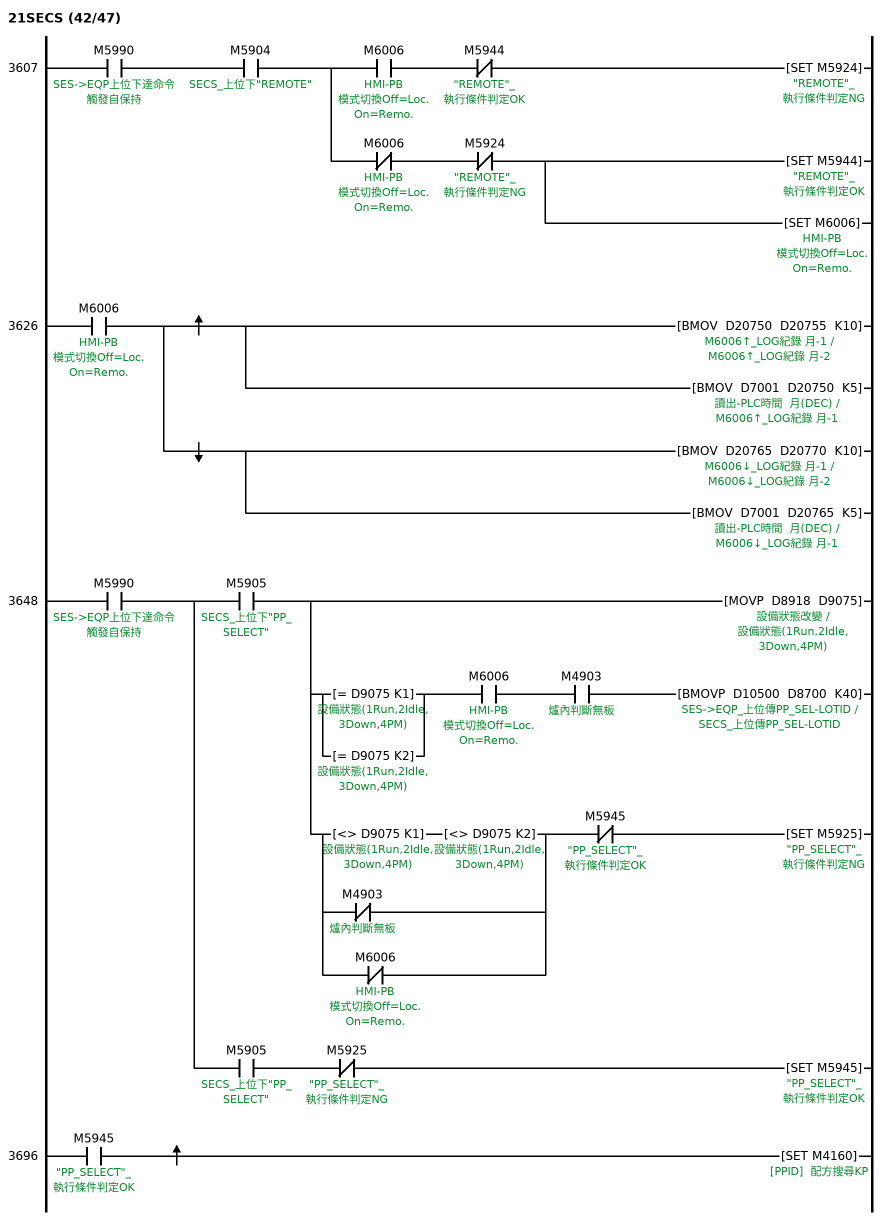
[picture p120: ladder of 21SECS, rungs at steps 3607 to 3696]
3607  LD      M5990  ; SES->EQP上位下達命令觸發自保持
      AND     M5904  ; SECS_上位下"REMOTE"
      MPS
      AND     M6006  ; HMI-PB  模式切換Off=Loc.On=Remo.
      ANI     M5944  ; "REMOTE"_執行條件判定OK
      SET     M5924  ; "REMOTE"_執行條件判定NG
        [note] "REMOTE CMD"
      MPP
      ANI     M6006  ; HMI-PB  模式切換Off=Loc.On=Remo.
      ANI     M5924  ; "REMOTE"_執行條件判定NG
      SET     M5944  ; "REMOTE"_執行條件判定OK
      SET     M6006  ; HMI-PB  模式切換Off=Loc.On=Remo.
3626  LD      M6006  ; HMI-PB  模式切換Off=Loc.On=Remo.
      MPS
      MEP
      BMOV    D20750 D20755 K10  ; M6006↑_LOG紀錄 月-1 / M6006↑_LOG紀錄 月-2
      BMOV    D7001 D20750 K5
      MPP
      MEF
      BMOV    D20765 D20770 K10  ; M6006↓_LOG紀錄 月-1 / M6006↓_LOG紀錄 月-2
      BMOV    D7001 D20765 K5
3648  LD      M5990  ; SES->EQP上位下達命令觸發自保持
      MPS
      AND     M5905  ; SECS_上位下"PP_SELECT"
      MOVP    D8918 D9075
        [note] "PP_SELECT CMD"
      MPS
      LD=     D9075 K1  ; 設備狀態(1Run,2Idle,3Down,4PM)
      OR=     D9075 K2  ; 設備狀態(1Run,2Idle,3Down,4PM)
      ANB
      AND     M6006  ; HMI-PB  模式切換Off=Loc.On=Remo.
      AND     M4903  ; 爐內判斷無板
      BMOVP   D10500 D8700 K40  ; SES->EQP_上位傳PP_SEL-LOTID / SECS_上位傳PP_SEL-LOTID
      MPP
      LD<>    D9075 K1  ; 設備狀態(1Run,2Idle,3Down,4PM)
      AND<>   D9075 K2  ; 設備狀態(1Run,2Idle,3Down,4PM)
      ORI     M4903  ; 爐內判斷無板
      ORI     M6006  ; HMI-PB  模式切換Off=Loc.On=Remo.
      ANB
      ANI     M5945  ; "PP_SELECT"_執行條件判定OK
      SET     M5925  ; "PP_SELECT"_執行條件判定NG
      MPP
      AND     M5905  ; SECS_上位下"PP_SELECT"
      ANI     M5925  ; "PP_SELECT"_執行條件判定NG
      SET     M5945  ; "PP_SELECT"_執行條件判定OK
3696  LD      M5945  ; "PP_SELECT"_執行條件判定OK
      MEP
      SET     M4160  ; [PPID]  配方搜尋KP
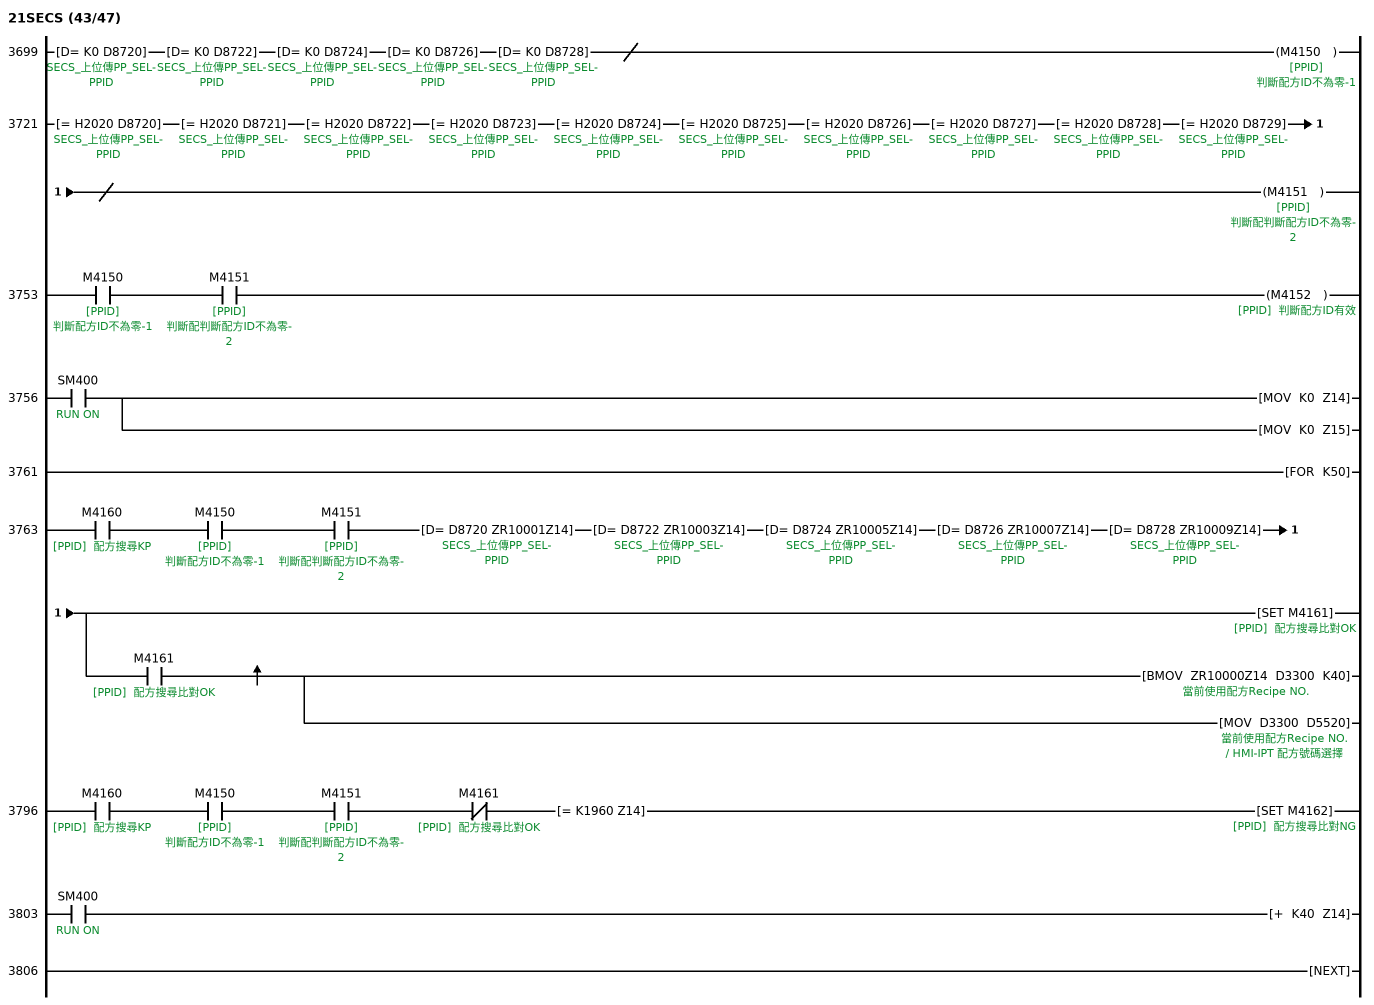
3699  LDD=    K0 D8720  ; SECS_上位傳PP_SEL-PPID
      ANDD=   K0 D8722  ; SECS_上位傳PP_SEL-PPID
      ANDD=   K0 D8724  ; SECS_上位傳PP_SEL-PPID
      ANDD=   K0 D8726  ; SECS_上位傳PP_SEL-PPID
      ANDD=   K0 D8728  ; SECS_上位傳PP_SEL-PPID
      INV
      OUT     M4150  ; [PPID]  判斷配方ID不為零-1
3721  LD=     H2020 D8720  ; SECS_上位傳PP_SEL-PPID
      AND=    H2020 D8721  ; SECS_上位傳PP_SEL-PPID
      AND=    H2020 D8722  ; SECS_上位傳PP_SEL-PPID
      AND=    H2020 D8723  ; SECS_上位傳PP_SEL-PPID
      AND=    H2020 D8724  ; SECS_上位傳PP_SEL-PPID
      AND=    H2020 D8725  ; SECS_上位傳PP_SEL-PPID
      AND=    H2020 D8726  ; SECS_上位傳PP_SEL-PPID
      AND=    H2020 D8727  ; SECS_上位傳PP_SEL-PPID
      AND=    H2020 D8728  ; SECS_上位傳PP_SEL-PPID
      AND=    H2020 D8729  ; SECS_上位傳PP_SEL-PPID
      INV
      OUT     M4151  ; [PPID]  判斷配判斷配方ID不為零-2
3753  LD      M4150  ; [PPID]  判斷配方ID不為零-1
      AND     M4151  ; [PPID]  判斷配判斷配方ID不為零-2
      OUT     M4152  ; [PPID]  判斷配方ID有效
3756  LD      SM400  ; RUN ON
      MOV     K0 Z14
      MOV     K0 Z15
3761  FOR     K50
3763  LD      M4160  ; [PPID]  配方搜尋KP
      AND     M4150  ; [PPID]  判斷配方ID不為零-1
      AND     M4151  ; [PPID]  判斷配判斷配方ID不為零-2
      ANDD=   D8720 ZR10001Z14  ; SECS_上位傳PP_SEL-PPID
      ANDD=   D8722 ZR10003Z14  ; SECS_上位傳PP_SEL-PPID
      ANDD=   D8724 ZR10005Z14  ; SECS_上位傳PP_SEL-PPID
      ANDD=   D8726 ZR10007Z14  ; SECS_上位傳PP_SEL-PPID
      ANDD=   D8728 ZR10009Z14  ; SECS_上位傳PP_SEL-PPID
      SET     M4161  ; [PPID]  配方搜尋比對OK
      AND     M4161  ; [PPID]  配方搜尋比對OK
      MEP
      BMOV    ZR10000Z14 D3300 K40
      MOV     D3300 D5520
3796  LD      M4160  ; [PPID]  配方搜尋KP
      AND     M4150  ; [PPID]  判斷配方ID不為零-1
      AND     M4151  ; [PPID]  判斷配判斷配方ID不為零-2
      ANI     M4161  ; [PPID]  配方搜尋比對OK
      AND=    K1960 Z14
      SET     M4162  ; [PPID]  配方搜尋比對NG
3803  LD      SM400  ; RUN ON
      +       K40 Z14
3806  NEXT
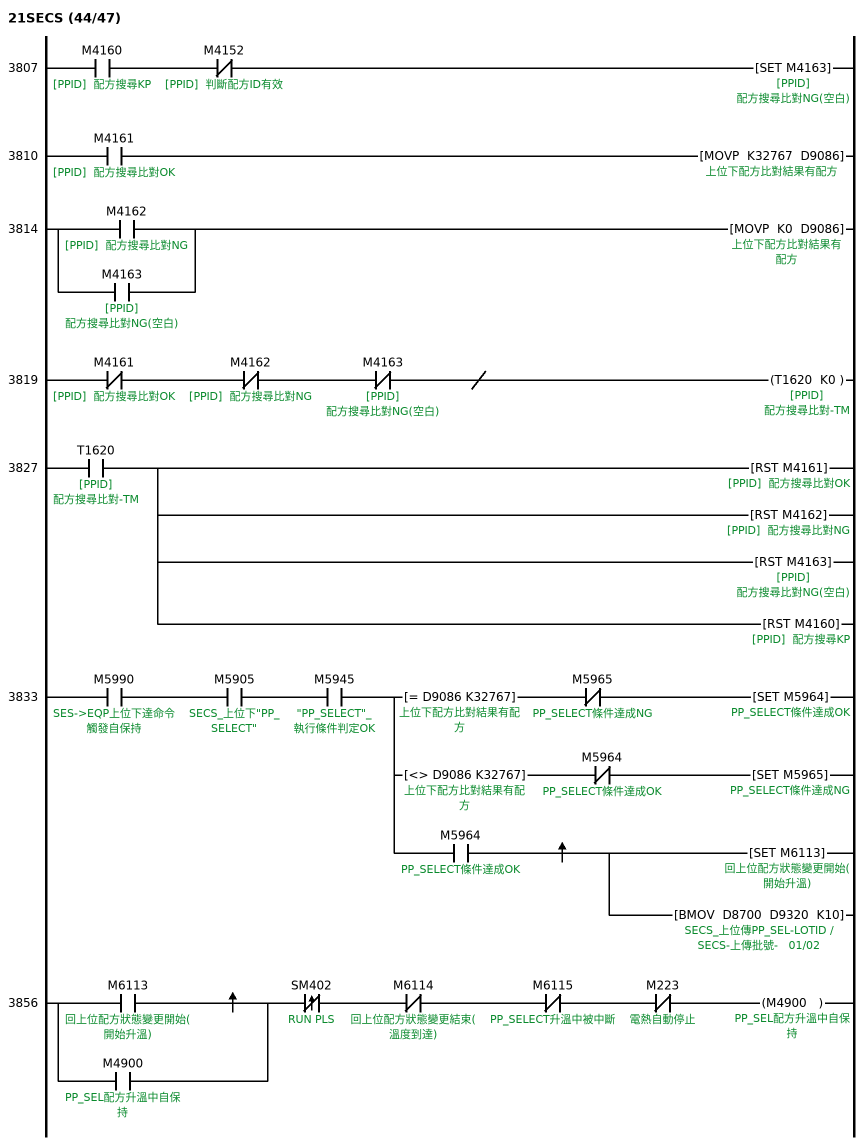
3807  LD      M4160  ; [PPID]  配方搜尋KP
      ANI     M4152  ; [PPID]  判斷配方ID有效
      SET     M4163  ; [PPID]  配方搜尋比對NG(空白)
3810  LD      M4161  ; [PPID]  配方搜尋比對OK
      MOVP    K32767 D9086
3814  LD      M4162  ; [PPID]  配方搜尋比對NG
      OR      M4163  ; [PPID]  配方搜尋比對NG(空白)
      MOVP    K0 D9086
3819  LDI     M4161  ; [PPID]  配方搜尋比對OK
      ANI     M4162  ; [PPID]  配方搜尋比對NG
      ANI     M4163  ; [PPID]  配方搜尋比對NG(空白)
      INV
      OUT     T1620 K0  ; [PPID]  配方搜尋比對-TM
3827  LD      T1620  ; [PPID]  配方搜尋比對-TM
      RST     M4161  ; [PPID]  配方搜尋比對OK
      RST     M4162  ; [PPID]  配方搜尋比對NG
      RST     M4163  ; [PPID]  配方搜尋比對NG(空白)
      RST     M4160  ; [PPID]  配方搜尋KP
3833  LD      M5990  ; SES->EQP上位下達命令觸發自保持
      AND     M5905  ; SECS_上位下"PP_SELECT"
      AND     M5945  ; "PP_SELECT"_執行條件判定OK
      MPS
      AND=    D9086 K32767  ; 上位下配方比對結果有配方
      ANI     M5965  ; PP_SELECT條件達成NG
      SET     M5964  ; PP_SELECT條件達成OK
      MRD
      AND<>   D9086 K32767  ; 上位下配方比對結果有配方
      ANI     M5964  ; PP_SELECT條件達成OK
      SET     M5965  ; PP_SELECT條件達成NG
      MPP
      AND     M5964  ; PP_SELECT條件達成OK
      MEP
      SET     M6113  ; 回上位配方狀態變更開始(開始升溫)
      BMOV    D8700 D9320 K10  ; SECS-上傳批號-   01/02
3856  LD      M6113  ; 回上位配方狀態變更開始(開始升溫)
      MEP
      OR      M4900  ; PP_SEL配方升溫中自保持
      ANDPI   SM402  ; RUN PLS
      ANI     M6114  ; 回上位配方狀態變更結束(溫度到達)
      ANI     M6115  ; PP_SELECT升溫中被中斷
      ANI     M223  ; 電熱自動停止
      OUT     M4900  ; PP_SEL配方升溫中自保持
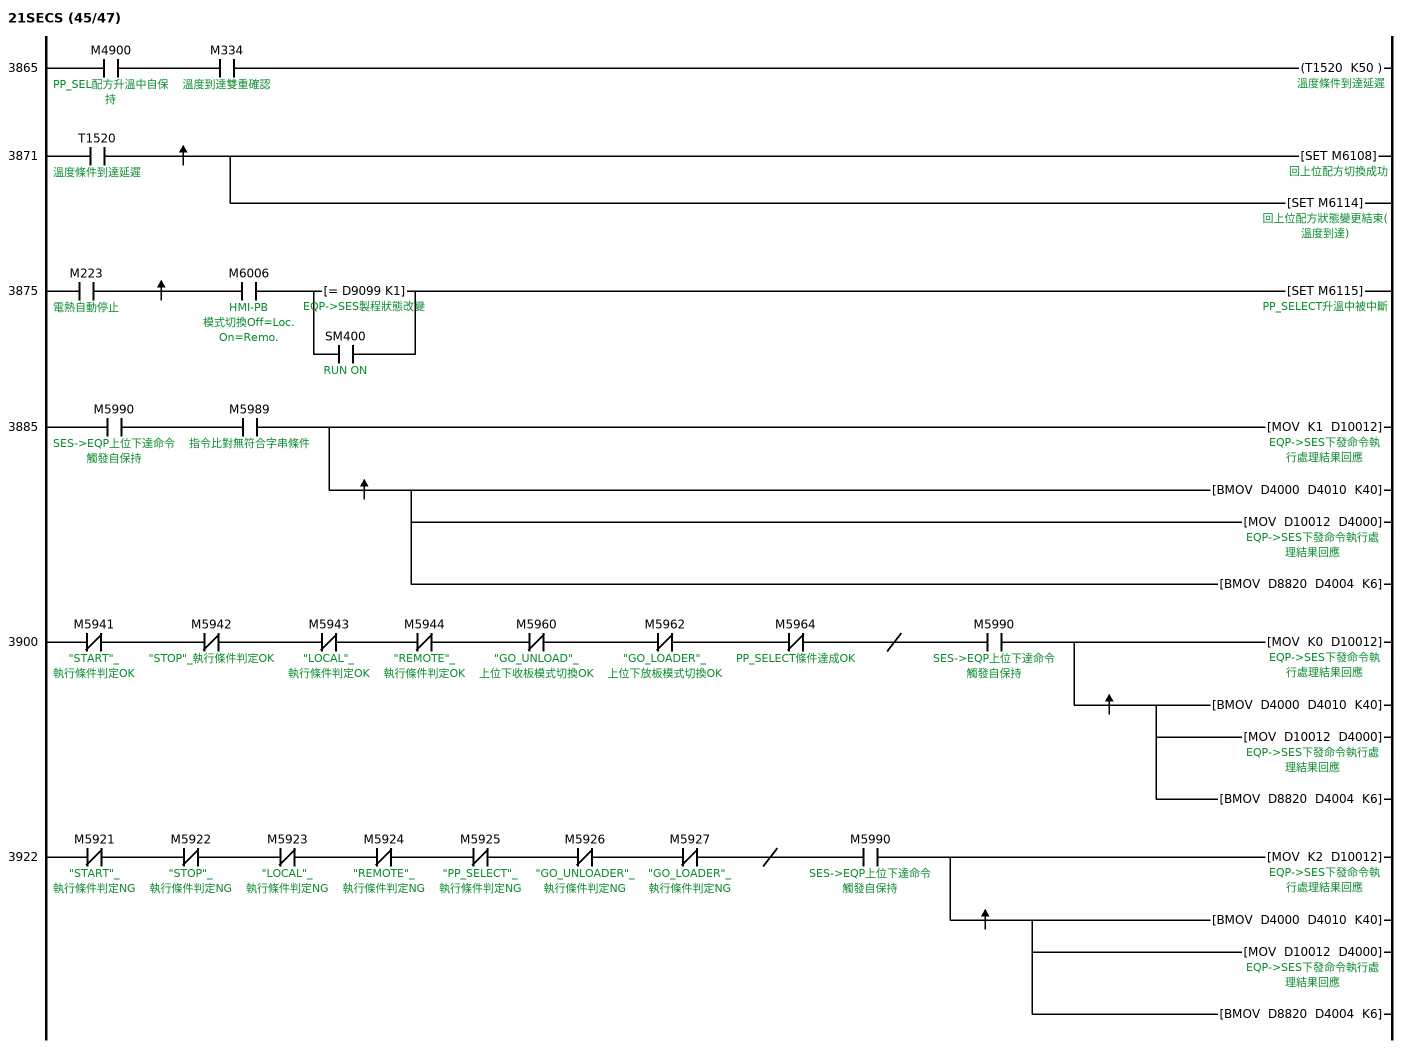
3865  LD      M4900  ; PP_SEL配方升溫中自保持
      AND     M334  ; 溫度到達雙重確認
      OUT     T1520 K50  ; 溫度條件到達延遲
3871  LD      T1520  ; 溫度條件到達延遲
      MEP
      SET     M6108  ; 回上位配方切換成功
      SET     M6114  ; 回上位配方狀態變更結束(溫度到達)
3875  LD      M223  ; 電熱自動停止
      MEP
      AND     M6006  ; HMI-PB  模式切換Off=Loc.On=Remo.
      LD=     D9099 K1  ; EQP->SES製程狀態改變
      OR      SM400  ; RUN ON
      ANB
      SET     M6115  ; PP_SELECT升溫中被中斷
3885  LD      M5990  ; SES->EQP上位下達命令觸發自保持
      AND     M5989  ; 指令比對無符合字串條件
      MOV     K1 D10012
      MEP
      BMOV    D4000 D4010 K40
      MOV     D10012 D4000
      BMOV    D8820 D4004 K6
3900  LDI     M5941  ; "START"_執行條件判定OK
      ANI     M5942  ; "STOP"_執行條件判定OK
      ANI     M5943  ; "LOCAL"_執行條件判定OK
      ANI     M5944  ; "REMOTE"_執行條件判定OK
      ANI     M5960  ; "GO_UNLOAD"_上位下收板模式切換OK
      ANI     M5962  ; "GO_LOADER"_上位下放板模式切換OK
      ANI     M5964  ; PP_SELECT條件達成OK
      INV
      AND     M5990  ; SES->EQP上位下達命令觸發自保持
      MOV     K0 D10012
      MEP
      BMOV    D4000 D4010 K40
      MOV     D10012 D4000
      BMOV    D8820 D4004 K6
3922  LDI     M5921  ; "START"_執行條件判定NG
      ANI     M5922  ; "STOP"_執行條件判定NG
      ANI     M5923  ; "LOCAL"_執行條件判定NG
      ANI     M5924  ; "REMOTE"_執行條件判定NG
      ANI     M5925  ; "PP_SELECT"_執行條件判定NG
      ANI     M5926  ; "GO_UNLOADER"_執行條件判定NG
      ANI     M5927  ; "GO_LOADER"_執行條件判定NG
      INV
      AND     M5990  ; SES->EQP上位下達命令觸發自保持
      MOV     K2 D10012
      MEP
      BMOV    D4000 D4010 K40
      MOV     D10012 D4000
      BMOV    D8820 D4004 K6
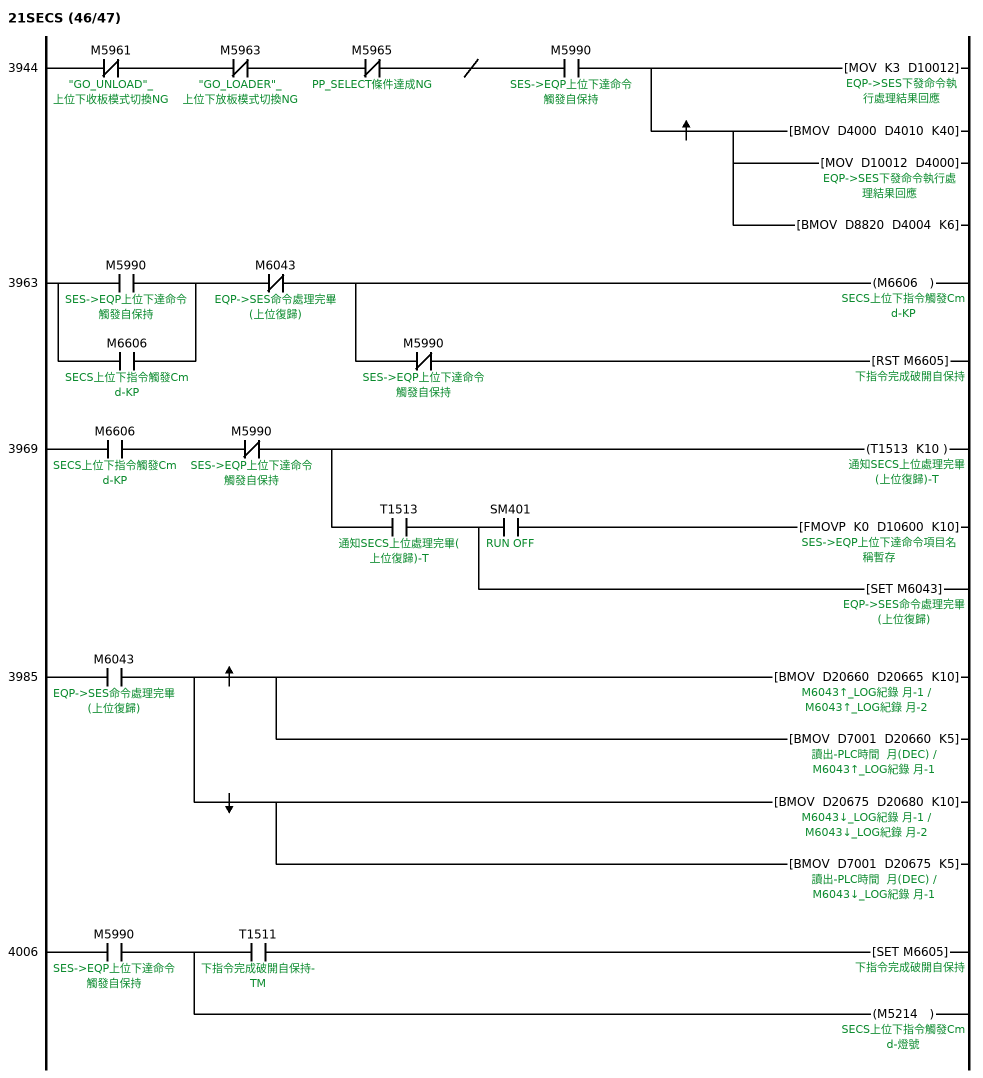
3944  LDI     M5961  ; "GO_UNLOAD"_上位下收板模式切換NG
      ANI     M5963  ; "GO_LOADER"_上位下放板模式切換NG
      ANI     M5965  ; PP_SELECT條件達成NG
      INV
      AND     M5990  ; SES->EQP上位下達命令觸發自保持
      MOV     K3 D10012
      MEP
      BMOV    D4000 D4010 K40
      MOV     D10012 D4000
      BMOV    D8820 D4004 K6
3963  LD      M5990  ; SES->EQP上位下達命令觸發自保持
      OR      M6606  ; SECS上位下指令觸發Cmd-KP
      ANI     M6043  ; EQP->SES命令處理完畢(上位復歸)
      OUT     M6606  ; SECS上位下指令觸發Cmd-KP
      ANI     M5990  ; SES->EQP上位下達命令觸發自保持
      RST     M6605  ; 下指令完成破開自保持
3969  LD      M6606  ; SECS上位下指令觸發Cmd-KP
      ANI     M5990  ; SES->EQP上位下達命令觸發自保持
      OUT     T1513 K10  ; 通知SECS上位處理完畢(上位復歸)-T
      AND     T1513  ; 通知SECS上位處理完畢(上位復歸)-T
      MPS
      AND     SM401  ; RUN OFF
      FMOVP   K0 D10600 K10
      MPP
      SET     M6043  ; EQP->SES命令處理完畢(上位復歸)
3985  LD      M6043  ; EQP->SES命令處理完畢(上位復歸)
      MPS
      MEP
      BMOV    D20660 D20665 K10  ; M6043↑_LOG紀錄 月-1 / M6043↑_LOG紀錄 月-2
      BMOV    D7001 D20660 K5
      MPP
      MEF
      BMOV    D20675 D20680 K10  ; M6043↓_LOG紀錄 月-1 / M6043↓_LOG紀錄 月-2
      BMOV    D7001 D20675 K5
4006  LD      M5990  ; SES->EQP上位下達命令觸發自保持
      MPS
      AND     T1511  ; 下指令完成破開自保持-TM
      SET     M6605  ; 下指令完成破開自保持
      MPP
      OUT     M5214  ; SECS上位下指令觸發Cmd-燈號
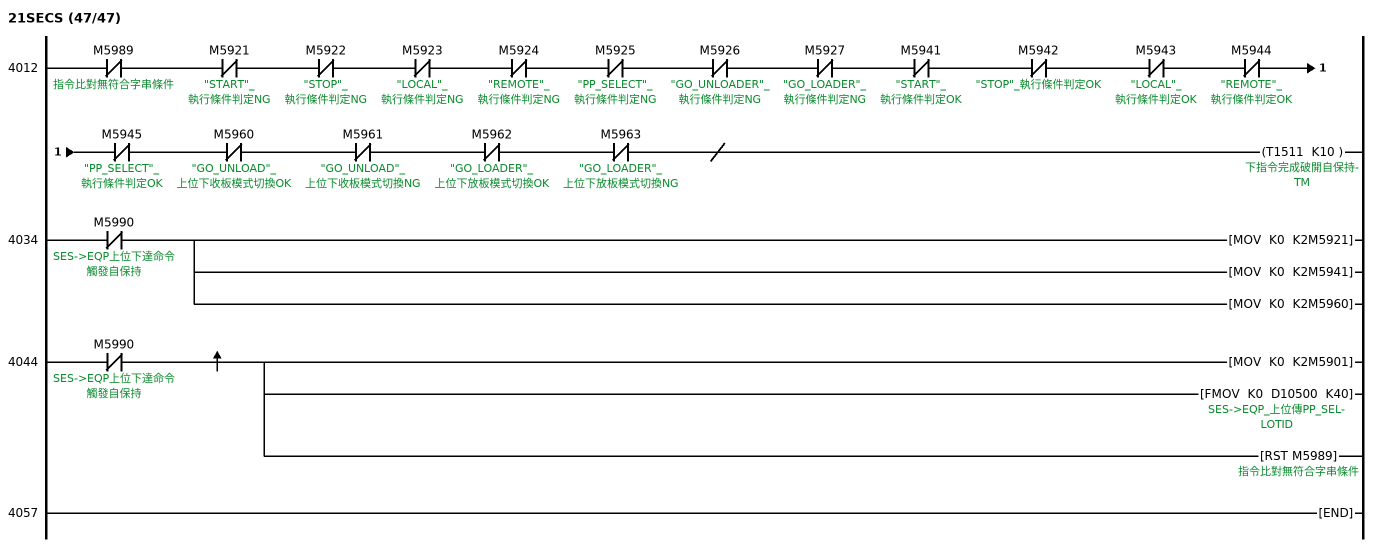
4012  LDI     M5989  ; 指令比對無符合字串條件
      ANI     M5921  ; "START"_執行條件判定NG
      ANI     M5922  ; "STOP"_執行條件判定NG
      ANI     M5923  ; "LOCAL"_執行條件判定NG
      ANI     M5924  ; "REMOTE"_執行條件判定NG
      ANI     M5925  ; "PP_SELECT"_執行條件判定NG
      ANI     M5926  ; "GO_UNLOADER"_執行條件判定NG
      ANI     M5927  ; "GO_LOADER"_執行條件判定NG
      ANI     M5941  ; "START"_執行條件判定OK
      ANI     M5942  ; "STOP"_執行條件判定OK
      ANI     M5943  ; "LOCAL"_執行條件判定OK
      ANI     M5944  ; "REMOTE"_執行條件判定OK
      ANI     M5945  ; "PP_SELECT"_執行條件判定OK
      ANI     M5960  ; "GO_UNLOAD"_上位下收板模式切換OK
      ANI     M5961  ; "GO_UNLOAD"_上位下收板模式切換NG
      ANI     M5962  ; "GO_LOADER"_上位下放板模式切換OK
      ANI     M5963  ; "GO_LOADER"_上位下放板模式切換NG
      INV
      OUT     T1511 K10  ; 下指令完成破開自保持-TM
4034  LDI     M5990  ; SES->EQP上位下達命令觸發自保持
      MOV     K0 K2M5921
      MOV     K0 K2M5941
      MOV     K0 K2M5960
4044  LDI     M5990  ; SES->EQP上位下達命令觸發自保持
      MEP
      MOV     K0 K2M5901
      FMOV    K0 D10500 K40
      RST     M5989  ; 指令比對無符合字串條件
4057  END
END_PROGRAM

// device comments not shown above
X4  ; 手動放板夾爪--放定點
X5  ; 手動放板夾爪--夾定點
X11  ; 取板完成位(連線)
X14  ; 下料旋臂長程中定點
X3C  ; 進料ROBOT左真空檢知
X7E  ; 印刷機出板要求
X332  ; FR1-DO(31)
X333  ; FR1-DO(32)
X334  ; FR1-DO(33)
X335  ; FR1-DO(34)
X336  ; FR1-DO(35)
X337  ; FR1-DO(36)
X338  ; FR1-DO(37)
X339  ; FR1-DO(38)
X33A  ; FR1-DO(39)
X33B  ; FR1-DO(40)
X33C  ; FR1-DO(41)
X33D  ; FR1-DO(42)
X33E  ; FR1-DO(43)
X33F  ; FR1-DO(44)
X340  ; FR1-DO(45)
X341  ; FR1-DO(46)
X342  ; FR1-DO(47)
X343  ; FR1-DO(48)
X344  ; FR1-DO(49)
X345  ; FR1-DO(50)
X346  ; FR1-DO(51)
X347  ; FR1-DO(52)
X348  ; FR1-DO(53)
X349  ; FR1-DO(54)
X34A  ; FR1-DO(55)
X34B  ; FR1-DO(56)
X34C  ; FR1-DO(57)
X34D  ; FR1-DO(58)
X34E  ; FR1-DO(59)
X34F  ; FR1-DO(60)
X350  ; FR1-DO(61)
X351  ; FR1-DO(62)
X352  ; FR1-DO(63)
X353  ; FR1-DO(64)
X354  ; FR1-DO(65)
X355  ; FR1-DO(66)
X356  ; FR1-DO(67)
X357  ; FR1-DO(68)
X358  ; FR1-DO(69)
X359  ; FR1-DO(70)
X35A  ; FR1-DO(71)
X35B  ; FR1-DO(72)
X35C  ; FR1-DO(73)
X35D  ; FR1-DO(74)
X35E  ; FR1-DO(75)
X35F  ; FR1-DO(76)
X360  ; FR1-DO(77)
X361  ; FR1-DO(78)
X362  ; FR1-DO(79)
X363  ; FR1-DO(80)
X364  ; FR1-DO(81)
X365  ; FR1-DO(82)
X366  ; FR1-DO(83)
X367  ; FR1-DO(84)
X368  ; FR1-DO(85)
X369  ; FR1-DO(86)
X36A  ; FR1-DO(87)
X36B  ; FR1-DO(88)
X36C  ; FR1-DO(89)
X36D  ; FR1-DO(90)
X36E  ; FR1-DO(91)
X36F  ; FR1-DO(92)
X370  ; FR1-DO(93)
X371  ; FR1-DO(94)
X372  ; FR1-DO(95)
X373  ; FR1-DO(96)
X374  ; FR1-DO(97)
X375  ; FR1-DO(98)
X376  ; FR1-DO(99)
X377  ; FR1-DO(100)
X378  ; FR1-DO(101)
X379  ; FR1-DO(102)
X37A  ; FR1-DO(103)
X37B  ; FR1-DO(104)
X37C  ; FR1-DO(105)
X37D  ; FR1-DO(106)
X37E  ; FR1-DO(107)
X37F  ; FR1-DO(108)
X0A03  ; Other station   DataLinkStatus
X1302  ; <印刷機>異常
Y10C  ; 進料連線--取板完
Y122  ; 進料ROBOT左真空SV
Y123  ; 進料ROBOT右真空SV
Y320  ; ROBOT GO HOME
Y330  ; TR1-DI(31)
Y331  ; TR1-DI(32)
Y332  ; TR1-DI(33)
Y333  ; TR1-DI(34)
Y334  ; TR1-DI(35)
Y335  ; TR1-DI(36)
Y336  ; TR1-DI(37)
Y337  ; TR1-DI(38)
Y338  ; TR1-DI(39)
Y339  ; TR1-DI(40)
Y33A  ; TR1-DI(41)
Y33B  ; TR1-DI(42)
Y33C  ; TR1-DI(43)
Y33D  ; TR1-DI(44)
Y33E  ; TR1-DI(45)
Y33F  ; TR1-DI(46)
Y340  ; TR1-DI(47)
Y341  ; TR1-DI(48)
Y342  ; TR1-DI(49)
Y343  ; TR1-DI(50)
Y344  ; TR1-DI(51)
Y345  ; TR1-DI(52)
Y346  ; TR1-DI(53)
Y347  ; TR1-DI(54)
Y348  ; TR1-DI(55)
Y349  ; TR1-DI(56)
Y34A  ; TR1-DI(57)
Y34B  ; TR1-DI(58)
Y34C  ; TR1-DI(59)
Y34D  ; TR1-DI(60)
Y34E  ; TR1-DI(61)
Y34F  ; TR1-DI(62)
Y350  ; TR1-DI(63)
Y351  ; TR1-DI(64)
Y352  ; TR1-DI(65)
Y353  ; TR1-DI(66)
Y354  ; TR1-DI(67)
Y355  ; TR1-DI(68)
Y356  ; TR1-DI(69)
Y357  ; TR1-DI(70)
Y358  ; TR1-DI(71)
Y359  ; TR1-DI(72)
Y35A  ; TR1-DI(73)
Y35B  ; TR1-DI(74)
Y35C  ; TR1-DI(75)
Y35D  ; TR1-DI(76)
Y35E  ; TR1-DI(77)
Y35F  ; TR1-DI(78)
Y360  ; TR1-DI(79)
Y361  ; TR1-DI(80)
Y362  ; TR1-DI(81)
Y363  ; TR1-DI(82)
Y364  ; TR1-DI(83)
Y365  ; TR1-DI(84)
Y366  ; TR1-DI(85)
Y367  ; TR1-DI(86)
Y368  ; TR1-DI(87)
Y369  ; TR1-DI(88)
Y36A  ; TR1-DI(89)
Y36B  ; TR1-DI(90)
Y36C  ; TR1-DI(91)
Y36D  ; TR1-DI(92)
Y36E  ; TR1-DI(93)
Y36F  ; TR1-DI(94)
Y370  ; TR1-DI(95)
Y371  ; TR1-DI(96)
Y372  ; TR1-DI(97)
Y373  ; TR1-DI(98)
Y374  ; TR1-DI(99)
Y375  ; TR1-DI(100)
Y376  ; TR1-DI(101)
Y377  ; TR1-DI(102)
Y378  ; TR1-DI(103)
Y379  ; TR1-DI(104)
Y37A  ; TR1-DI(105)
Y37B  ; TR1-DI(106)
Y37C  ; TR1-DI(107)
Y37D  ; TR1-DI(108)
Y37E  ; TR1-DI(109)
Y37F  ; TR1-DI(110)
M40  ; 手動放板側邊上料_放板PB
M42  ; 夾爪開爪腳踏開關_側邊上料使用PB
M55  ; 板材尺寸連線/本機模式PB
M70  ; 昇降上昇位置教導設定PB
M71  ; 昇降上等待位置教導設定PB
M73  ; 昇降下降位置教導設定PB
M76  ; 下料鼓風機自動
M79  ; 下料鼓風機手動
M140  ; 手動放板側邊上料_放板燈
M141  ; 手動放板側邊上料_夾板燈
M182  ; 進料照明開
M185  ; 出料照明開
M190  ; 上料掉板後原點復歸
M191  ; 上料掉板後原點復歸STOP
M221  ; 搬移停止
M234  ; 自動模式鏈條拉緊PLS
M237  ; 上料夾爪可伸出KP
M316  ; 開機鏈條張力自動拉緊
M317  ; 鏈條張力拉緊KP
M318  ; 主傳動步進拉緊
M324  ; 電熱溫度到達KP
M325  ; 電熱溫度到達計時
M326  ; 開機計時24小時到
M327  ; 油壓張力檢知
M332  ; 進料輸送停止
M333  ; 進料輸送減速KP
M335  ; 升溫中狀態
M375  ; 手動放板側邊上料_放板
M376  ; 手動放板側邊上料_夾板
M377  ; 手動上板PB4指示燈
M439  ; 進料ROBOT禁止回原點
M514  ; 下料旋臂長程中定點
M552  ; 進料集塵鼓風機手動運轉
M553  ; 出料集塵鼓風機手動運轉
M554  ; 進出料集塵鼓風機自動運轉
M595  ; #06 風車PB
M596  ; #07 風車PB
M597  ; #08 風車PB
M598  ; #09 風車PB
M599  ; #10 風車PB
M600  ; #11 風車PB
M601  ; #12 風車PB
M602  ; #13 風車PB
M603  ; #14 風車PB
M604  ; #15 風車PB
M605  ; #16 風車PB
M606  ; #17 風車PB
M615  ; #06 電熱PB
M616  ; #07 電熱PB
M617  ; #08 電熱PB
M618  ; #09 電熱PB
M619  ; #10 電熱PB
M620  ; #11 電熱PB
M621  ; #12 電熱PB
M622  ; #13 電熱PB
M623  ; #14 電熱PB
M624  ; #15 電熱PB
M625  ; #16 電熱PB
M626  ; #17 電熱PB
M700  ; SECS_USE清除進板訊號
M701  ; SECS_USE進板訊號ON
M725  ; #06 風車訊號
M726  ; #07 風車訊號
M727  ; #08 風車訊號
M728  ; #09 風車訊號
M729  ; #10 風車訊號
M730  ; #11 風車訊號
M731  ; #12 風車訊號
M732  ; #13 風車訊號
M733  ; #14 風車訊號
M734  ; #15 風車訊號
M735  ; #16 風車訊號
M736  ; #17 風車訊號
M785  ; #06 電熱訊號
M786  ; #07 電熱訊號
M787  ; #08 電熱訊號
M788  ; #09 電熱訊號
M789  ; #10 電熱訊號
M790  ; #11 電熱訊號
M791  ; #12 電熱訊號
M792  ; #13 電熱訊號
M793  ; #14 電熱訊號
M794  ; #15 電熱訊號
M795  ; #16 電熱訊號
M796  ; #17 電熱訊號
M805  ; 上料夾爪短程縮回KP
M825  ; #06 溫度到達KP
M826  ; #07 溫度到達KP
M827  ; #08 溫度到達KP
M828  ; #09 溫度到達KP
M829  ; #10 溫度到達KP
M830  ; #11 溫度到達KP
M831  ; #12 溫度到達KP
M832  ; #13 溫度到達KP
M833  ; #14 溫度到達KP
M834  ; #15 溫度到達KP
M835  ; #16 溫度到達KP
M836  ; #17 溫度到達KP
M1010  ; SECS_USE指令比對正確
M1011  ; PP_SELECT條件達成
M1304  ; 進料段無板
M1305  ; 進料定位有板
M1518  ; 風車停止備用1PLS
M1519  ; 風車停止備用2PLS
M1605  ; #06 電熱AL2 超溫
M1606  ; #07 電熱AL2 超溫
M1607  ; #08 電熱AL2 超溫
M1615  ; 冷卻段電熱AL2 超溫
M1621  ; #06 電熱OTP 超溫
M1622  ; #07 電熱OTP 超溫
M1623  ; #08 電熱OTP 超溫
M1637  ; #06 風車過載
M1638  ; #07 風車過載
M1639  ; #08 風車過載
M1653  ; #06 低溫警報
M1654  ; #07 低溫警報
M1655  ; #08 低溫警報
M4704  ; 生產片數到達
M4713  ; 拍板馬達伺服運轉逾時異常
M4716  ; 拍板馬達伺服內極限
M4717  ; 拍板馬達伺服外極限
M4917  ; 刪除配方名稱
M4920  ; 入口計數
M4921  ; 出口計數
M4922  ; 爐內限制異常
M4923  ; 出口計數
M4925  ; 卡板不警報
M4930  ; 點燈運轉KP
M4931  ; 點燈停止
M4932  ; 上位下啟動訊號
M4933  ; PP_SELECT點燈用保持
M4934  ; 上位允許放板START
M4935  ; 上位下暫停進板
M4936  ; HMI-Show_SEC模式未START
M4937  ; 上位要儲存配方
M4943  ; 上位下GO_REMOTE
M4944  ; 上位下GO-LOCAL
M4945  ; 上位允許放板START保持
M4950  ; 點燈中請稍待指示
M4951  ; 熄點燈冷卻中請稍待指示
M4953  ; 熄燈OK狀態
M4956  ; 輸送機停止熄燈
M4990  ; 密碼ENT
M4992  ; 密碼ENT Keep
M4993  ; 參數設定取消PB
M4994  ; 參數設定取消PLS
M4996  ; 離線測試用
M4999  ; 回上位生產停止
M5004  ; ##未完成生產片數到達
M5034  ; 輸送運轉未加熱完成
M5075  ; 回上位生產完成保持
M5076  ; IDLE-   FLAG
M5101  ; 三色紅燈
M5102  ; 三色綠燈
M5106  ; 未知?測試用
M5203  ; 未知?測試用
M5204  ; 上位允許放板START
M5205  ; 上位停止放板並清出料號
M5206  ; 上位下配方和啟動輸送和點燈
M5207  ; 上位切換成GO-REMOTE
M5208  ; 上位切換成GO-LOCAL
M5209  ; 上位下暫停進板
M5210  ; 上位下恢復進板
M5213  ; 上位下指令觸發bit
M5215  ; Barcod啟動固定式完成
M5216  ; 上位字串比對不對(開始,停止,配方)
M5217  ; 門,(1)(2),PPID,配方名稱比對不對
M5314  ; 配方刪除
M5315  ; 配方儲存
M5316  ; 呼叫Q的配方
M5317  ; 比對配方用
M5318  ; 自動
M5319  ; 手動
M5320  ; FX機台狀態改變
M5321  ; 自動啟動
M5322  ; 程式結束
M5323  ; 緊急停止開關
M5325  ; 對話視窗關閉
M5326  ; 配方新增
M5327  ; 配方修改
M5328  ; 配方刪除
M5329  ; 機構異常警報
M5347  ; 配方Barcode掃描
M5348  ; 工單輸入
M5349  ; Barcod啟動固定式
M5350  ; Bey Pass PB
M5351  ; 自動PB
M5352  ; 連線開放OP控制
M5353  ; 確認(101頁)人機SET
M5354  ; 確認(102頁)人機SET
M5410  ; [ES-01] GREEN_  LiGHT   OFF
M5411  ; [ES-01] GREEN_  LiGHT   ON
M5412  ; [ES-01] GREEN_  LiGHT   FLASH
M5413  ; [ES-01] RED_    LiGHT   OFF
M5414  ; [ES-01] RED_    LiGHT   ON
M5415  ; [ES-01] RED_    LiGHT   FLASH
M5416  ; [ES-01] YELLOW_ LiGHT   OFF
M5417  ; [ES-01] YELLOW_ LiGHT   ON
M5418  ; [ES-01] YELLOW_ LiGHT   FLASH
M5928  ; "STC"_執行條件判定NG
M5929  ; "BUZZER"_執行條件判定NG
M5946  ; "GO_UNLOADER"_執行條件判定OK
M5947  ; "GO_LOADER"_執行條件判定OK
M5948  ; "STC"_執行條件判定OK
M5949  ; "BUZZER"_執行條件判定OK
M5970  ; MES收板模式初始化動作中
M5972  ; MES放板模式初始化動作中
M6140  ; 要求上位回讀工單板號右爐
M6141  ; 要求上位回讀工單右爐
M6231  ; 上位要儲存配方
M6600  ; SECS上位下指令觸發Cmd-KP
M6607  ; Host刪除配方自保持
M6608  ; Host刪除配方自清除保持
M6610  ; 比對M700~M715都等於零
M6611  ; 比對M716~M731都等於零
M6820  ; 比對GO-REMOTE字串不對
M6821  ; 名稱GO-LOCAL比對不對
M6822  ; 比對RESUME字串不對
M6823  ; 比對PPID字串不對
M6824  ; 比對PAUSE字串不對
M6825  ; 比對START字串不對
M6826  ; 比對STOP字串不對
M6827  ; 比對PP_SELECT字串不對
M6854  ; 機台再IDEL
M6860  ; 機台不在可生產狀態
M6861  ; 下STOP 機台不再READY/EXECUTING
M6862  ; 下PP_SELECT 機台不在待機中(IDLE)
M6863  ; 設備沒再暫停狀態
M6864  ; 機台不再START 狀態
M6865  ; 機台狀態不對
M6866  ; 設備沒再LOCAL狀態
M6867  ; 設備沒再REMOTE狀態
M6999  ; 三色綠燈
M7001  ; 三色紅燈
M7012  ; 回應HOST要儲存配方同步
M7014  ; 回應HOST刪除配方同步
M7600  ; RUN ON
L3804  ; 第05站  CC-LINK 異常
L3805  ; 第06站  CC-LINK 異常
L3806  ; 第07站  CC-LINK 異常
L3807  ; 第08站  CC-LINK 異常
L3808  ; 第09站  CC-LINK 異常
L3809  ; 第10站  CC-LINK 異常
L3810  ; 第11站  CC-LINK 異常
L3811  ; 第12站  CC-LINK 異常
L3812  ; 第13站  CC-LINK 異常
L3813  ; 第14站  CC-LINK 異常
L3814  ; 第15站  CC-LINK 異常
L3815  ; 第16站  CC-LINK 異常
T8  ; 上料伺服自動復歸次數未到計時
T11  ; 上料伺服自動復歸計時
T12  ; 上料手臂夾爪夾自動延遲
T13  ; 上料昇降伺服運轉延遲
T16  ; 昇降上昇位置教導延遲
T17  ; 昇降上等待位置教導延遲
T19  ; 昇降下降位置教導延遲
T39  ; 下料鼓風機自動停止
T47  ; 進料集塵鼓風機PB延遲
T48  ; 出料集塵鼓風機PB延遲
T49  ; 集塵鼓風機運轉停止延遲
T54  ; 進料段無板延遲
T56  ; ROBOT外部循環啟動計時
T68  ; 進料輸送減速光電延遲
T75  ; 油壓馬達送電前進10秒
T105  ; #06 風車PB延遲
T106  ; #07 風車PB延遲
T107  ; #08 風車PB延遲
T108  ; #09 風車PB延遲
T109  ; #10 風車PB延遲
T110  ; #11 風車PB延遲
T111  ; #12 風車PB延遲
T112  ; #13 風車PB延遲
T113  ; #14 風車PB延遲
T114  ; #15 風車PB延遲
T115  ; #16 風車PB延遲
T116  ; #17 風車PB延遲
T125  ; #06 電熱PB延遲
T126  ; #07 電熱PB延遲
T127  ; #08 電熱PB延遲
T128  ; #09 電熱PB延遲
T129  ; #10 電熱PB延遲
T130  ; #11 電熱PB延遲
T131  ; #12 電熱PB延遲
T132  ; #13 電熱PB延遲
T133  ; #14 電熱PB延遲
T134  ; #15 電熱PB延遲
T135  ; #16 電熱PB延遲
T136  ; #17 電熱PB延遲
T139  ; #17 低溫警報
T145  ; #06 低溫警報
T146  ; #07 低溫警報
T147  ; #08 低溫警報
T148  ; #09 低溫警報
T149  ; #10 低溫警報
T150  ; #11 低溫警報
T151  ; #12 低溫警報
T152  ; #13 低溫警報
T159  ; 進料輸送夾爪夾板異常延遲
T163  ; 進料輸送垂直異常延遲
T164  ; 進料輸送水平異常延遲
T165  ; 上料夾爪長程伸異常延遲
T166  ; 上料夾爪長程縮異常延遲
T186  ; 油壓馬達運轉計時
T188  ; 進料輸送運轉逾時
T190  ; 進料輸送掉板異常延遲
T191  ; 上料夾爪掉板異常延遲
T196  ; 進料空氣壓力異常延時
T200  ; 進料輸送停止時間延遲
T204  ; 進料ROBOT左真空檢知異常TM
T205  ; 進料ROBOT右真空檢知異常TM
T208  ; 手動上板檢知光電異常TM
T400  ; #01 風車INV運轉計時
T401  ; #02 風車INV運轉計時
T402  ; #03 風車INV運轉計時
T403  ; #04 風車INV運轉計時
T404  ; #05 風車INV運轉計時
T405  ; #06 風車INV運轉計時
T406  ; #07 風車INV運轉計時
T407  ; #08 風車INV運轉計時
T408  ; #09 風車INV運轉計時
T409  ; #10 風車INV運轉計時
T410  ; #11 風車INV運轉計時
T411  ; #12 風車INV運轉計時
T412  ; #13 風車INV運轉計時
T413  ; #14 風車INV運轉計時
T414  ; #15 風車INV運轉計時
T415  ; #16 風車INV運轉計時
T420  ; 進料風車INV運轉計時
T421  ; 出料風車INV運轉計時
T425  ; 進料輸送INV運轉計時
T1010  ; [ES-01] GREEN_  LiGHT   OFF
T1011  ; [ES-01] GREEN_  LiGHT   ON
T1013  ; [ES-01] RED_    LiGHT   OFF
T1014  ; [ES-01] RED_    LiGHT   ON
T1016  ; [ES-01] YELLOW_ LiGHT   OFF
T1017  ; [ES-01] YELLOW_ LiGHT   ON
T1055  ; SECS_USE開機延遲一秒
T1101  ; EQP->SES控制模式切換(On/Off)-TM
T1102  ; EQP->SES機台狀態改變-TM
T1103  ; EQP->SES操作模式自動/手動-TM
T1104  ; EQP->SES當前使用配方變更-TM
T1105  ; EQP->SES回上位新增配方-TM
T1106  ; EQP->SES回上位刪除配方-TM
T1107  ; EQP->SES回上位修改配方-TM
T1108  ; 回上位配方切換成功-TM
T1109  ; EQP>SES Panel   Start-TM
T1110  ; EQP>SES Panel   End-TM
T1111  ; EQP->SES回上位  LotStart-TM
T1112  ; EQP->SES回上位  LotEnd-TM
T1113  ; 回上位配方狀態變更開始(升溫)-TM
T1114  ; 回上位配方狀態變更結束(到達)-TM
T1115  ; PP_SELECT升溫中被中斷-TM
T1127  ; 夾爪放定點延時
T1201  ; 下指令完成破開自保持-TM
T1202  ; SECS上位下指令觸發Cmd復歸-TM
T1203  ; 通知SECS上位處理完畢(上位復歸)-T
T1275  ; 回上位生產完成延遲
C0  ; 自動模式計數24小時
D22  ; 昇降伺服設定參數
D23  ; 昇降伺服異常碼
D24  ; 昇降伺服異常碼
D35  ; 年*10000
D37  ; 月*100
D39  ; 人機時間年月日
D40  ; 電熱溫度到達計時sec
D41  ; 進料輸送停止時間延遲
D81  ; 爐內無板延遲時間切換SV(RUN->IDLE
D150  ; 人機參數密碼
D163  ; 1槽風速CH5
D164  ; 2槽風速CH6
D165  ; 3槽風速CH7
D166  ; 4槽風速CH8
D167  ; 5槽風速CH9
D170  ; 1靜置風速CH3
D171  ; 2靜置風速CH4
D172  ; 1冷卻風速CH10
D173  ; 2冷卻風速CH11
D222  ; 上料手臂取板位置暫存
D249  ; 上料手臂夾爪現在位置換算板寬
D251  ; 上料手臂夾爪現在位置
D253  ; 上料手臂夾爪伺服現在速度
D261  ; 上料手臂夾爪運轉速度設定
D263  ; 上料手臂夾爪JOG速度值
D265  ; 上料手臂夾爪設定位置設定值
D267  ; 上料手臂夾爪原點位置設定值
D297  ; 總生產量Hi
D301  ; 本班產量履歷2
D302  ; 本班產量履歷3
D303  ; 本班產量履歷4
D304  ; 本班產量履歷5
D305  ; 本班產量履歷6
D306  ; 本班產量履歷7
D307  ; 本班產量履歷8
D308  ; 本班產量履歷9
D309  ; 本班產量履歷10
D310  ; 本班產量履歷11
D311  ; 本班產量履歷12
D312  ; 本班產量履歷13
D313  ; 本班產量履歷14
D314  ; 本班產量履歷15
D315  ; 本班產量履歷16
D316  ; 本班產量履歷17
D317  ; 本班產量履歷18
D318  ; 本班產量履歷19
D319  ; 本班產量履歷20
D320  ; 本班產量履歷21
D321  ; 本班產量履歷22
D322  ; 本班產量履歷23
D323  ; 本班產量履歷24
D324  ; 本班產量履歷25
D331  ; 現在時間時分2
D332  ; 現在時間時分3
D333  ; 現在時間時分4
D334  ; 現在時間時分5
D335  ; 現在時間時分6
D336  ; 現在時間時分7
D337  ; 現在時間時分8
D338  ; 現在時間時分9
D339  ; 現在時間時分10
D340  ; 現在時間時分11
D341  ; 現在時間時分12
D342  ; 現在時間時分13
D343  ; 現在時間時分14
D344  ; 現在時間時分15
D345  ; 現在時間時分16
D346  ; 現在時間時分17
D347  ; 現在時間時分18
D348  ; 現在時間時分19
D349  ; 現在時間時分20
D350  ; 現在時間時分21
D351  ; 現在時間時分22
D352  ; 現在時間時分23
D353  ; 現在時間時分24
D354  ; 現在時間時分25
D395  ; 月保養時間現在值
D397  ; 季保養時間現在值
D399  ; 年保養時間現在值
D405  ; PLC=>SV6
D406  ; PLC=>SV7
D407  ; PLC=>SV8
D408  ; PLC=>SV9
D409  ; PLC=>SV10
D425  ; PV6=>PLC
D426  ; PV7=>PLC
D427  ; PV8=>PLC
D428  ; PV9=>PLC
D429  ; PV10=>PLC
D440  ; SV1=>PLC
D441  ; SV2=>PLC
D442  ; SV3=>PLC
D443  ; SV4=>PLC
D444  ; SV5=>PLC
D445  ; SV6=>PLC
D446  ; SV7=>PLC
D447  ; SV8=>PLC
D448  ; SV9=>PLC
D449  ; SV10=>PLC
D548  ; 中心拍板現在位置換算板寬
D549  ; 中心拍板現在位置換算板寬
D550  ; 中心拍板夾爪現在位置
D551  ; 中心拍板夾爪現在位置
D552  ; 中心拍板夾爪伺服現在速度
D553  ; 中心拍板夾爪伺服現在速度
D554  ; 中心拍板伺服異常碼
D560  ; 中心拍板運轉速度設定
D561  ; 中心拍板運轉速度設定
D562  ; 中心拍板JOG速度值
D563  ; 中心拍板JOG速度值
D564  ; 中心拍板設定位置設定值
D565  ; 中心拍板設定位置設定值
D566  ; 中心拍板原點位置設定值
D567  ; 中心拍板原點位置設定值
D641  ; 烘烤時間SEC
D701  ; 月保養時數
D711  ; 季保養時數
D721  ; 年保養時數
D809  ; 排氣風壓檢知異常警報
D859  ; 排氣風壓檢知異常警報暫存
D1001  ; 系統時間年月日00
D1002  ; 系統時間年月日01
D1003  ; 系統時間年月日01
D1004  ; 系統時間年月日02
D1005  ; 系統時間年月日02
D1006  ; 系統時間年月日03
D1007  ; 系統時間年月日03
D1008  ; 系統時間年月日04
D1009  ; 系統時間年月日04
D1010  ; 系統時間年月日05
D1011  ; 系統時間年月日05
D1012  ; 系統時間年月日06
D1013  ; 系統時間年月日06
D1014  ; 系統時間年月日07
D1015  ; 系統時間年月日07
D1016  ; 系統時間年月日08
D1017  ; 系統時間年月日08
D1018  ; 系統時間年月日09
D1019  ; 系統時間年月日09
D1020  ; 系統時間年月日10
D1021  ; 系統時間年月日10
D1022  ; 系統時間年月日11
D1023  ; 系統時間年月日11
D1024  ; 系統時間年月日12
D1025  ; 系統時間年月日12
D1026  ; 系統時間年月日13
D1027  ; 系統時間年月日13
D1028  ; 系統時間年月日14
D1029  ; 系統時間年月日14
D1030  ; 系統時間年月日15
D1031  ; 系統時間年月日15
D1032  ; 系統時間年月日16
D1033  ; 系統時間年月日16
D1034  ; 系統時間年月日17
D1035  ; 系統時間年月日17
D1036  ; 系統時間年月日18
D1037  ; 系統時間年月日18
D1038  ; 系統時間年月日19
D1039  ; 系統時間年月日19
D1040  ; 系統時間年月日20
D1041  ; 系統時間年月日20
D1042  ; 系統時間年月日21
D1043  ; 系統時間年月日21
D1044  ; 系統時間年月日22
D1045  ; 系統時間年月日22
D1046  ; 系統時間年月日23
D1047  ; 系統時間年月日23
D1048  ; 系統時間年月日24
D1049  ; 系統時間年月日24
D1200  ; 第01槽電熱實際溫度PV
D1201  ; 第02槽電熱實際溫度PV
D1202  ; 第03槽電熱實際溫度PV
D1203  ; 第04槽電熱實際溫度PV
D1204  ; 第05槽電熱實際溫度PV
D1205  ; 第06槽電熱實際溫度PV
D1206  ; 第07槽電熱實際溫度PV
D1207  ; 第08槽電熱實際溫度PV
D1208  ; 第09槽電熱實際溫度PV
D1209  ; 第10槽電熱實際溫度PV
D1210  ; 第11槽電熱實際溫度PV
D1211  ; 第12槽電熱實際溫度PV
D1230  ; 第1槽溫度記錄次數
D1232  ; 第1槽溫度累加值
D1234  ; 第1槽溫度均值
D1240  ; 第1槽低溫警報
D1242  ; 第1槽超溫警報
D1244  ; 第1槽平均值低溫警報
D1246  ; 第1槽平均值超溫警報
D1250  ; 第12槽溫度記錄次數
D1252  ; 第12槽溫度累加值
D1254  ; 第12槽溫度均值
D1260  ; 第12槽低溫警報
D1262  ; 第12槽超溫警報
D1264  ; 第12槽平均值低溫警報
D1266  ; 第1槽平均值超溫警報
D1300  ; 第01槽電熱溫度設定SV
D1301  ; 第02槽電熱溫度設定SV
D1302  ; 第03槽電熱溫度設定SV
D1303  ; 第04槽電熱溫度設定SV
D1304  ; 第05槽電熱溫度設定SV
D1305  ; 第06槽電熱溫度設定SV
D1306  ; 第07槽電熱溫度設定SV
D1307  ; 第08槽電熱溫度設定SV
D1308  ; 第09槽電熱溫度設定SV
D1309  ; 第10槽電熱溫度設定SV
D1310  ; 第11槽電熱溫度設定SV
D1311  ; 第12槽電熱溫度設定SV
D1325  ; 第06槽電熱溫度設定SV-2
D1326  ; 第07槽電熱溫度設定SV-2
D1327  ; 第08槽電熱溫度設定SV-2
D1328  ; 第09槽電熱溫度設定SV-2
D1329  ; 第10槽電熱溫度設定SV-2
D1330  ; 第11槽電熱溫度設定SV-2
D1331  ; 第12槽電熱溫度設定SV-2
D1345  ; 第06槽電熱溫度設定SV+2
D1346  ; 第07槽電熱溫度設定SV+2
D1347  ; 第08槽電熱溫度設定SV+2
D1348  ; 第09槽電熱溫度設定SV+2
D1349  ; 第10槽電熱溫度設定SV+2
D1350  ; 第11槽電熱溫度設定SV+2
D1351  ; 第12槽電熱溫度設定SV+2
D2002  ; TR1 ROBOT取板點(補償)Z
D2009  ; TR1 ROBOT放板點(補償)Y
D2010  ; TR1 ROBOT放板點(補償)Z
D2100  ; TR1(R30)ROBOT運轉速率_1%~100%
D2101  ; TR1(R31)手臂取板點(補償)X
D2102  ; TR1(R32)手臂取板點(補償)Y
D2103  ; TR1(R33)手臂取板點(補償)Z
D2104  ; TR1(R34)手臂取板點(補償)角度
D2105  ; TR1(R35)手臂放板點(補償)X
D2106  ; TR1(R36)手臂放板點(補償)Y
D2107  ; TR1(R37)手臂放板點(補償)Z
D2108  ; TR1(R38)手臂放板點(補償)角度
D2109  ; TR1(R39)板長尺寸偏差量(0.1mm)
D2110  ; TR1(R40)
D2111  ; TR1(R41)
D2112  ; TR1(R42)
D2113  ; TR1(R43)
D2114  ; TR1(R44)
D2115  ; TR1(R45)
D2503  ; 人機手臂取板點(補償)Z
D2505  ; 人機手臂放板點(補償)Y
D2506  ; 人機手臂放板點(補償)Z
D3302  ; 當前使用配方RecipeID#04/03
D3303  ; 當前使用配方RecipeID#06/05
D3304  ; 當前使用配方RecipeID#08/07
D3305  ; 當前使用配方RecipeID#10/09
D3306  ; 當前使用配方RecipeID#12/11
D3307  ; 當前使用配方RecipeID#14/13
D3308  ; 當前使用配方RecipeID#16/15
D3309  ; 當前使用配方RecipeID#18/17
D3310  ; 當前使用配方RecipeID#20/19
D3311  ; 當前使用配方RecipeID#22/21
D3312  ; 當前使用配方RecipeID#24/23
D3313  ; 當前使用配方RecipeID#26/25
D3314  ; 當前使用配方RecipeID#28/27
D3315  ; 當前使用配方RecipeID#30/29
D3316  ; 當前使用配方RecipeID#32/31
D3317  ; 當前使用配方RecipeID#34/33
D3318  ; 當前使用配方RecipeID#36/35
D3319  ; 當前使用配方RecipeID#38/37
D3320  ; 當前使用配方RecipeID#40/39
D3322  ; 當前使用配方第02槽電熱設定
D3323  ; 當前使用配方第03槽電熱設定
D3324  ; 當前使用配方第04槽電熱設定
D3325  ; 當前使用配方第05槽電熱設定
D3326  ; 當前使用配方第06槽電熱設定
D3327  ; 當前使用配方第07槽電熱設定
D3328  ; 當前使用配方第08槽電熱設定
D3329  ; 當前使用配方第09槽電熱設定
D3330  ; 當前使用配方第10槽電熱設定
D3331  ; 當前使用配方第11槽電熱設定
D3332  ; 當前使用配方第12槽電熱設定
D3339  ; 當前使用配方烘烤時間(分)
D3390  ; HMI-編輯RecipeID#22/21
D3391  ; HMI-編輯RecipeID#24/23
D3392  ; HMI-編輯RecipeID#26/25
D3393  ; HMI-編輯RecipeID#28/27
D3394  ; HMI-編輯RecipeID#30/29
D3395  ; HMI-編輯RecipeID#32/31
D3396  ; HMI-編輯RecipeID#34/33
D3397  ; HMI-編輯RecipeID#36/35
D3398  ; HMI-編輯RecipeID#38/37
D3399  ; HMI-編輯RecipeID#40/39
D3405  ; HMI-編輯第06槽電熱設定
D3406  ; HMI-編輯第07槽電熱設定
D3407  ; HMI-編輯第08槽電熱設定
D3408  ; HMI-編輯第09槽電熱設定
D3409  ; HMI-編輯第10槽電熱設定
D3410  ; HMI-編輯第11槽電熱設定
D3411  ; HMI-編輯第12槽電熱設定
D3414  ; HMI-編輯板材尺寸寬度設定
D3420  ; HMI-編輯爐內烘烤時間計算-2(秒)
D3422  ; HMI-編輯爐內烘烤時間計算-2(分)
D4940  ; SP.SOC OPEN指令控制數據
D4944  ; SP.SOC SND指令結束元件
D4950  ; SP.SOC  SND指令控制數據
D4952  ; SP.SOC  RCV指令控制數據
D4954  ; SP.SOC  CLOSE指令控制數據
D5105  ; ATMA->GP板長mm
D5106  ; ATMA->GP板寬mm
D5140  ; CHANNEL
D5142  ; INDEX
D5144  ; Channel Range
D5200  ; 第01槽  風速值
D5202  ; 第02槽  風速值
D5204  ; 第03槽  風速值
D5206  ; 第04槽  風速值
D5208  ; 第05槽  風速值
D5300  ; 參數X1  01
D5302  ; 參數X1  02
D5304  ; 參數X1  03
D5306  ; 參數X1  04
D5308  ; 參數X1  05
D5400  ; 參數Y1  01
D5402  ; 參數Y1  02
D5404  ; 參數Y1  03
D5406  ; 參數Y1  04
D5408  ; 參數Y1  05
D5508  ; [ED-02] 配方異動型態
D5514  ; 配方組別計算-2-(1)
D10070  ; 比對START字串
D10071  ; 比對STOP字串
D10072  ; 比對PP_SELECT字串
D10074  ; 比對配方名稱為零可儲存位址
D10076  ; 名稱有一樣的是更新=50要新增
D10077  ; 比對PAUSE字串
D10078  ; 比對RESUME字串
D10081  ; 上位下配方比對結果
D10083  ; 上位下的組別右門(比對出來的)
D10084  ; 名稱GO-LOCAL比對結果
D10085  ; 名稱PPID比對結果
D10086  ; 上位下配方比對結果
D10087  ; 上位下的組別左門(比對出來的)
D10590  ; SECS_上位下START指令
D10625  ; SECS_上位下STOP指令
D10640  ; SECS_上位下RESUME指令
D10675  ; SECS_上位下PPID指令
D10676  ; SECS_上位下PPID指令
D10900  ; "ST"ART
D10901  ; ST"AR"T
D10902  ; STAR"T"
D10910  ; "ST"OP
D10911  ; ST"OP"
D10920  ; "PP"_SELECT
D10921  ; PP"_S"ELECT
D10922  ; PP_S"EL"ECT
D10923  ; PP_SEL"EC"T
D10924  ; PP_SELEC"T"
D10930  ; "RE"MOTE
D10931  ; RE"MO"TE
D10932  ; REMO"TE"
D10940  ; "LO"CAL
D10941  ; LO"CA"L
D10942  ; LOCA"L"
D10945  ; "PP"ID
D10946  ; PP"ID"
D10950  ; "PA"USE
D10951  ; PA"US"E
D10952  ; PAUS"E"
D10960  ; "RE"SUME
D10961  ; RE"SU"ME
D10962  ; RESU"ME"
D13517  ; 第01槽電熱實際溫度PV(FLT)
D13519  ; 第02槽電熱實際溫度PV(FLT)
D13521  ; 第03槽電熱實際溫度PV(FLT)
D13523  ; 第04槽電熱實際溫度PV(FLT)
D13525  ; 第05槽電熱實際溫度PV(FLT)
D13526  ; 第01槽風壓檢知PV(FLT)
D13527  ; 第01槽風壓檢知PV(FLT)
D13528  ; 第02槽風壓檢知PV(FLT)
D13529  ; 第02槽風壓檢知PV(FLT)
D13530  ; 第03槽風壓檢知PV(FLT)
D13531  ; 第03槽風壓檢知PV(FLT)
D13532  ; 第04槽風壓檢知PV(FLT)
D13533  ; 第04槽風壓檢知PV(FLT)
D13534  ; 第05槽風壓檢知PV(FLT)
D13535  ; 第05槽風壓檢知PV(FLT)
D13607  ; 查詢配方內容板材尺寸寬度設定
D20001  ; M6002↑_LOG紀錄 日-1
D20002  ; M6002↑_LOG紀錄 時-1
D20003  ; M6002↑_LOG紀錄 分-1
D20004  ; M6002↑_LOG紀錄 秒-1
D20006  ; M6002↑_LOG紀錄 日-2
D20007  ; M6002↑_LOG紀錄 時-2
D20008  ; M6002↑_LOG紀錄 分-2
D20009  ; M6002↑_LOG紀錄 秒-2
D20010  ; M6002↑_LOG紀錄 月-3
D20011  ; M6002↑_LOG紀錄 日-3
D20012  ; M6002↑_LOG紀錄 時-3
D20013  ; M6002↑_LOG紀錄 分-3
D20014  ; M6002↑_LOG紀錄 秒-3
D20016  ; M6002↓_LOG紀錄 日-1
D20017  ; M6002↓_LOG紀錄 時-1
D20018  ; M6002↓_LOG紀錄 分-1
D20019  ; M6002↓_LOG紀錄 秒-1
D20021  ; M6002↓_LOG紀錄 日-2
D20022  ; M6002↓_LOG紀錄 時-2
D20023  ; M6002↓_LOG紀錄 分-2
D20024  ; M6002↓_LOG紀錄 秒-2
D20025  ; M6002↓_LOG紀錄 月-3
D20026  ; M6002↓_LOG紀錄 日-3
D20027  ; M6002↓_LOG紀錄 時-3
D20028  ; M6002↓_LOG紀錄 分-3
D20029  ; M6002↓_LOG紀錄 秒-3
D20031  ; M9101↑_LOG紀錄 日-1
D20032  ; M9101↑_LOG紀錄 時-1
D20033  ; M9101↑_LOG紀錄 分-1
D20034  ; M9101↑_LOG紀錄 秒-1
D20036  ; M9101↑_LOG紀錄 日-2
D20037  ; M9101↑_LOG紀錄 時-2
D20038  ; M9101↑_LOG紀錄 分-2
D20039  ; M9101↑_LOG紀錄 秒-2
D20040  ; M9101↑_LOG紀錄 月-3
D20041  ; M9101↑_LOG紀錄 日-3
D20042  ; M9101↑_LOG紀錄 時-3
D20043  ; M9101↑_LOG紀錄 分-3
D20044  ; M9101↑_LOG紀錄 秒-3
D20046  ; M9101↓_LOG紀錄 日-1
D20047  ; M9101↓_LOG紀錄 時-1
D20048  ; M9101↓_LOG紀錄 分-1
D20049  ; M9101↓_LOG紀錄 秒-1
D20051  ; M9101↓_LOG紀錄 日-2
D20052  ; M9101↓_LOG紀錄 時-2
D20053  ; M9101↓_LOG紀錄 分-2
D20054  ; M9101↓_LOG紀錄 秒-2
D20055  ; M9101↓_LOG紀錄 月-3
D20056  ; M9101↓_LOG紀錄 日-3
D20057  ; M9101↓_LOG紀錄 時-3
D20058  ; M9101↓_LOG紀錄 分-3
D20059  ; M9101↓_LOG紀錄 秒-3
D20061  ; M6005↑_LOG紀錄 日-1
D20062  ; M6005↑_LOG紀錄 時-1
D20063  ; M6005↑_LOG紀錄 分-1
D20064  ; M6005↑_LOG紀錄 秒-1
D20066  ; M6005↑_LOG紀錄 日-2
D20067  ; M6005↑_LOG紀錄 時-2
D20068  ; M6005↑_LOG紀錄 分-2
D20069  ; M6005↑_LOG紀錄 秒-2
D20070  ; M6005↑_LOG紀錄 月-3
D20071  ; M6005↑_LOG紀錄 日-3
D20072  ; M6005↑_LOG紀錄 時-3
D20073  ; M6005↑_LOG紀錄 分-3
D20074  ; M6005↑_LOG紀錄 秒-3
D20076  ; M6005↓_LOG紀錄 日-1
D20077  ; M6005↓_LOG紀錄 時-1
D20078  ; M6005↓_LOG紀錄 分-1
D20079  ; M6005↓_LOG紀錄 秒-1
D20081  ; M6005↓_LOG紀錄 日-2
D20082  ; M6005↓_LOG紀錄 時-2
D20083  ; M6005↓_LOG紀錄 分-2
D20084  ; M6005↓_LOG紀錄 秒-2
D20085  ; M6005↓_LOG紀錄 月-3
D20086  ; M6005↓_LOG紀錄 日-3
D20087  ; M6005↓_LOG紀錄 時-3
D20088  ; M6005↓_LOG紀錄 分-3
D20089  ; M6005↓_LOG紀錄 秒-3
D20091  ; M6101↑_LOG紀錄 日-1
D20092  ; M6101↑_LOG紀錄 時-1
D20093  ; M6101↑_LOG紀錄 分-1
D20094  ; M6101↑_LOG紀錄 秒-1
D20096  ; M6101↑_LOG紀錄 日-2
D20097  ; M6101↑_LOG紀錄 時-2
D20098  ; M6101↑_LOG紀錄 分-2
D20099  ; M6101↑_LOG紀錄 秒-2
D20100  ; M6101↑_LOG紀錄 月-3
D20101  ; M6101↑_LOG紀錄 日-3
D20102  ; M6101↑_LOG紀錄 時-3
D20103  ; M6101↑_LOG紀錄 分-3
D20104  ; M6101↑_LOG紀錄 秒-3
D20106  ; M6101↓_LOG紀錄 日-1
D20107  ; M6101↓_LOG紀錄 時-1
D20108  ; M6101↓_LOG紀錄 分-1
D20109  ; M6101↓_LOG紀錄 秒-1
D20111  ; M6101↓_LOG紀錄 日-2
D20112  ; M6101↓_LOG紀錄 時-2
D20113  ; M6101↓_LOG紀錄 分-2
D20114  ; M6101↓_LOG紀錄 秒-2
D20115  ; M6101↓_LOG紀錄 月-3
D20116  ; M6101↓_LOG紀錄 日-3
D20117  ; M6101↓_LOG紀錄 時-3
D20118  ; M6101↓_LOG紀錄 分-3
D20119  ; M6101↓_LOG紀錄 秒-3
D20121  ; M6102↑_LOG紀錄 日-1
D20122  ; M6102↑_LOG紀錄 時-1
D20123  ; M6102↑_LOG紀錄 分-1
D20124  ; M6102↑_LOG紀錄 秒-1
D20126  ; M6102↑_LOG紀錄 日-2
D20127  ; M6102↑_LOG紀錄 時-2
D20128  ; M6102↑_LOG紀錄 分-2
D20129  ; M6102↑_LOG紀錄 秒-2
D20130  ; M6102↑_LOG紀錄 月-3
D20131  ; M6102↑_LOG紀錄 日-3
D20132  ; M6102↑_LOG紀錄 時-3
D20133  ; M6102↑_LOG紀錄 分-3
D20134  ; M6102↑_LOG紀錄 秒-3
D20136  ; M6102↓_LOG紀錄 日-1
D20137  ; M6102↓_LOG紀錄 時-1
D20138  ; M6102↓_LOG紀錄 分-1
D20139  ; M6102↓_LOG紀錄 秒-1
D20141  ; M6102↓_LOG紀錄 日-2
D20142  ; M6102↓_LOG紀錄 時-2
D20143  ; M6102↓_LOG紀錄 分-2
D20144  ; M6102↓_LOG紀錄 秒-2
D20145  ; M6102↓_LOG紀錄 月-3
D20146  ; M6102↓_LOG紀錄 日-3
D20147  ; M6102↓_LOG紀錄 時-3
D20148  ; M6102↓_LOG紀錄 分-3
D20149  ; M6102↓_LOG紀錄 秒-3
D20151  ; M6015↑_LOG紀錄 日-1
D20152  ; M6015↑_LOG紀錄 時-1
D20153  ; M6015↑_LOG紀錄 分-1
D20154  ; M6015↑_LOG紀錄 秒-1
D20156  ; M6015↑_LOG紀錄 日-2
D20157  ; M6015↑_LOG紀錄 時-2
D20158  ; M6015↑_LOG紀錄 分-2
D20159  ; M6015↑_LOG紀錄 秒-2
D20160  ; M6015↑_LOG紀錄 月-3
D20161  ; M6015↑_LOG紀錄 日-3
D20162  ; M6015↑_LOG紀錄 時-3
D20163  ; M6015↑_LOG紀錄 分-3
D20164  ; M6015↑_LOG紀錄 秒-3
D20166  ; M6015↓_LOG紀錄 日-1
D20167  ; M6015↓_LOG紀錄 時-1
D20168  ; M6015↓_LOG紀錄 分-1
D20169  ; M6015↓_LOG紀錄 秒-1
D20171  ; M6015↓_LOG紀錄 日-2
D20172  ; M6015↓_LOG紀錄 時-2
D20173  ; M6015↓_LOG紀錄 分-2
D20174  ; M6015↓_LOG紀錄 秒-2
D20175  ; M6015↓_LOG紀錄 月-3
D20176  ; M6015↓_LOG紀錄 日-3
D20177  ; M6015↓_LOG紀錄 時-3
D20178  ; M6015↓_LOG紀錄 分-3
D20179  ; M6015↓_LOG紀錄 秒-3
D20181  ; M6009↑_LOG紀錄 日-1
D20182  ; M6009↑_LOG紀錄 時-1
D20183  ; M6009↑_LOG紀錄 分-1
D20184  ; M6009↑_LOG紀錄 秒-1
D20186  ; M6009↑_LOG紀錄 日-2
D20187  ; M6009↑_LOG紀錄 時-2
D20188  ; M6009↑_LOG紀錄 分-2
D20189  ; M6009↑_LOG紀錄 秒-2
D20190  ; M6009↑_LOG紀錄 月-3
D20191  ; M6009↑_LOG紀錄 日-3
D20192  ; M6009↑_LOG紀錄 時-3
D20193  ; M6009↑_LOG紀錄 分-3
D20194  ; M6009↑_LOG紀錄 秒-3
D20196  ; M6009↓_LOG紀錄 日-1
D20197  ; M6009↓_LOG紀錄 時-1
D20198  ; M6009↓_LOG紀錄 分-1
D20199  ; M6009↓_LOG紀錄 秒-1
D20201  ; M6009↓_LOG紀錄 日-2
D20202  ; M6009↓_LOG紀錄 時-2
D20203  ; M6009↓_LOG紀錄 分-2
D20204  ; M6009↓_LOG紀錄 秒-2
D20205  ; M6009↓_LOG紀錄 月-3
D20206  ; M6009↓_LOG紀錄 日-3
D20207  ; M6009↓_LOG紀錄 時-3
D20208  ; M6009↓_LOG紀錄 分-3
D20209  ; M6009↓_LOG紀錄 秒-3
D20211  ; M6138↑_LOG紀錄 日-1
D20212  ; M6138↑_LOG紀錄 時-1
D20213  ; M6138↑_LOG紀錄 分-1
D20214  ; M6138↑_LOG紀錄 秒-1
D20216  ; M6138↑_LOG紀錄 日-2
D20217  ; M6138↑_LOG紀錄 時-2
D20218  ; M6138↑_LOG紀錄 分-2
D20219  ; M6138↑_LOG紀錄 秒-2
D20220  ; M6138↑_LOG紀錄 月-3
D20221  ; M6138↑_LOG紀錄 日-3
D20222  ; M6138↑_LOG紀錄 時-3
D20223  ; M6138↑_LOG紀錄 分-3
D20224  ; M6138↑_LOG紀錄 秒-3
D20226  ; M6138↓_LOG紀錄 日-1
D20227  ; M6138↓_LOG紀錄 時-1
D20228  ; M6138↓_LOG紀錄 分-1
D20229  ; M6138↓_LOG紀錄 秒-1
D20231  ; M6138↓_LOG紀錄 日-2
D20232  ; M6138↓_LOG紀錄 時-2
D20233  ; M6138↓_LOG紀錄 分-2
D20234  ; M6138↓_LOG紀錄 秒-2
D20235  ; M6138↓_LOG紀錄 月-3
D20236  ; M6138↓_LOG紀錄 日-3
D20237  ; M6138↓_LOG紀錄 時-3
D20238  ; M6138↓_LOG紀錄 分-3
D20239  ; M6138↓_LOG紀錄 秒-3
D20241  ; M6238↑_LOG紀錄 日-1
D20242  ; M6238↑_LOG紀錄 時-1
D20243  ; M6238↑_LOG紀錄 分-1
D20244  ; M6238↑_LOG紀錄 秒-1
D20246  ; M6238↑_LOG紀錄 日-2
D20247  ; M6238↑_LOG紀錄 時-2
D20248  ; M6238↑_LOG紀錄 分-2
D20249  ; M6238↑_LOG紀錄 秒-2
D20250  ; M6238↑_LOG紀錄 月-3
D20251  ; M6238↑_LOG紀錄 日-3
D20252  ; M6238↑_LOG紀錄 時-3
D20253  ; M6238↑_LOG紀錄 分-3
D20254  ; M6238↑_LOG紀錄 秒-3
D20256  ; M6238↓_LOG紀錄 日-1
D20257  ; M6238↓_LOG紀錄 時-1
D20258  ; M6238↓_LOG紀錄 分-1
D20259  ; M6238↓_LOG紀錄 秒-1
D20261  ; M6238↓_LOG紀錄 日-2
D20262  ; M6238↓_LOG紀錄 時-2
D20263  ; M6238↓_LOG紀錄 分-2
D20264  ; M6238↓_LOG紀錄 秒-2
D20265  ; M6238↓_LOG紀錄 月-3
D20266  ; M6238↓_LOG紀錄 日-3
D20267  ; M6238↓_LOG紀錄 時-3
D20268  ; M6238↓_LOG紀錄 分-3
D20269  ; M6238↓_LOG紀錄 秒-3
D20271  ; M6103↑_LOG紀錄 日-1
D20272  ; M6103↑_LOG紀錄 時-1
D20273  ; M6103↑_LOG紀錄 分-1
D20274  ; M6103↑_LOG紀錄 秒-1
D20276  ; M6103↑_LOG紀錄 日-2
D20277  ; M6103↑_LOG紀錄 時-2
D20278  ; M6103↑_LOG紀錄 分-2
D20279  ; M6103↑_LOG紀錄 秒-2
D20280  ; M6103↑_LOG紀錄 月-3
D20281  ; M6103↑_LOG紀錄 日-3
D20282  ; M6103↑_LOG紀錄 時-3
D20283  ; M6103↑_LOG紀錄 分-3
D20284  ; M6103↑_LOG紀錄 秒-3
D20286  ; M6103↓_LOG紀錄 日-1
D20287  ; M6103↓_LOG紀錄 時-1
D20288  ; M6103↓_LOG紀錄 分-1
D20289  ; M6103↓_LOG紀錄 秒-1
D20291  ; M6103↓_LOG紀錄 日-2
D20292  ; M6103↓_LOG紀錄 時-2
D20293  ; M6103↓_LOG紀錄 分-2
D20294  ; M6103↓_LOG紀錄 秒-2
D20295  ; M6103↓_LOG紀錄 月-3
D20296  ; M6103↓_LOG紀錄 日-3
D20297  ; M6103↓_LOG紀錄 時-3
D20298  ; M6103↓_LOG紀錄 分-3
D20299  ; M6103↓_LOG紀錄 秒-3
D20301  ; M6109↑_LOG紀錄 日-1
D20302  ; M6109↑_LOG紀錄 時-1
D20303  ; M6109↑_LOG紀錄 分-1
D20304  ; M6109↑_LOG紀錄 秒-1
D20306  ; M6109↑_LOG紀錄 日-2
D20307  ; M6109↑_LOG紀錄 時-2
D20308  ; M6109↑_LOG紀錄 分-2
D20309  ; M6109↑_LOG紀錄 秒-2
D20310  ; M6109↑_LOG紀錄 月-3
D20311  ; M6109↑_LOG紀錄 日-3
D20312  ; M6109↑_LOG紀錄 時-3
D20313  ; M6109↑_LOG紀錄 分-3
D20314  ; M6109↑_LOG紀錄 秒-3
D20316  ; M6109↓_LOG紀錄 日-1
D20317  ; M6109↓_LOG紀錄 時-1
D20318  ; M6109↓_LOG紀錄 分-1
D20319  ; M6109↓_LOG紀錄 秒-1
D20321  ; M6109↓_LOG紀錄 日-2
D20322  ; M6109↓_LOG紀錄 時-2
D20323  ; M6109↓_LOG紀錄 分-2
D20324  ; M6109↓_LOG紀錄 秒-2
D20325  ; M6109↓_LOG紀錄 月-3
D20326  ; M6109↓_LOG紀錄 日-3
D20327  ; M6109↓_LOG紀錄 時-3
D20328  ; M6109↓_LOG紀錄 分-3
D20329  ; M6109↓_LOG紀錄 秒-3
D20331  ; M6110↑_LOG紀錄 日-1
D20332  ; M6110↑_LOG紀錄 時-1
D20333  ; M6110↑_LOG紀錄 分-1
D20334  ; M6110↑_LOG紀錄 秒-1
D20336  ; M6110↑_LOG紀錄 日-2
D20337  ; M6110↑_LOG紀錄 時-2
D20338  ; M6110↑_LOG紀錄 分-2
D20339  ; M6110↑_LOG紀錄 秒-2
D20340  ; M6110↑_LOG紀錄 月-3
D20341  ; M6110↑_LOG紀錄 日-3
D20342  ; M6110↑_LOG紀錄 時-3
D20343  ; M6110↑_LOG紀錄 分-3
D20344  ; M6110↑_LOG紀錄 秒-3
D20346  ; M6110↓_LOG紀錄 日-1
D20347  ; M6110↓_LOG紀錄 時-1
D20348  ; M6110↓_LOG紀錄 分-1
D20349  ; M6110↓_LOG紀錄 秒-1
D20351  ; M6110↓_LOG紀錄 日-2
D20352  ; M6110↓_LOG紀錄 時-2
D20353  ; M6110↓_LOG紀錄 分-2
D20354  ; M6110↓_LOG紀錄 秒-2
D20355  ; M6110↓_LOG紀錄 月-3
D20356  ; M6110↓_LOG紀錄 日-3
D20357  ; M6110↓_LOG紀錄 時-3
D20358  ; M6110↓_LOG紀錄 分-3
D20359  ; M6110↓_LOG紀錄 秒-3
D20361  ; M6233↑_LOG紀錄 日-1
D20362  ; M6233↑_LOG紀錄 時-1
D20363  ; M6233↑_LOG紀錄 分-1
D20364  ; M6233↑_LOG紀錄 秒-1
D20366  ; M6233↑_LOG紀錄 日-2
D20367  ; M6233↑_LOG紀錄 時-2
D20368  ; M6233↑_LOG紀錄 分-2
D20369  ; M6233↑_LOG紀錄 秒-2
D20370  ; M6233↑_LOG紀錄 月-3
D20371  ; M6233↑_LOG紀錄 日-3
D20372  ; M6233↑_LOG紀錄 時-3
D20373  ; M6233↑_LOG紀錄 分-3
D20374  ; M6233↑_LOG紀錄 秒-3
D20376  ; M6233↓_LOG紀錄 日-1
D20377  ; M6233↓_LOG紀錄 時-1
D20378  ; M6233↓_LOG紀錄 分-1
D20379  ; M6233↓_LOG紀錄 秒-1
D20381  ; M6233↓_LOG紀錄 日-2
D20382  ; M6233↓_LOG紀錄 時-2
D20383  ; M6233↓_LOG紀錄 分-2
D20384  ; M6233↓_LOG紀錄 秒-2
D20385  ; M6233↓_LOG紀錄 月-3
D20386  ; M6233↓_LOG紀錄 日-3
D20387  ; M6233↓_LOG紀錄 時-3
D20388  ; M6233↓_LOG紀錄 分-3
D20389  ; M6233↓_LOG紀錄 秒-3
D20391  ; M6024↑_LOG紀錄 日-1
D20392  ; M6024↑_LOG紀錄 時-1
D20393  ; M6024↑_LOG紀錄 分-1
D20394  ; M6024↑_LOG紀錄 秒-1
D20396  ; M6024↑_LOG紀錄 日-2
D20397  ; M6024↑_LOG紀錄 時-2
D20398  ; M6024↑_LOG紀錄 分-2
D20399  ; M6024↑_LOG紀錄 秒-2
D20400  ; M6024↑_LOG紀錄 月-3
D20401  ; M6024↑_LOG紀錄 日-3
D20402  ; M6024↑_LOG紀錄 時-3
D20403  ; M6024↑_LOG紀錄 分-3
D20404  ; M6024↑_LOG紀錄 秒-3
D20406  ; M6024↓_LOG紀錄 日-1
D20407  ; M6024↓_LOG紀錄 時-1
D20408  ; M6024↓_LOG紀錄 分-1
D20409  ; M6024↓_LOG紀錄 秒-1
D20411  ; M6024↓_LOG紀錄 日-2
D20412  ; M6024↓_LOG紀錄 時-2
D20413  ; M6024↓_LOG紀錄 分-2
D20414  ; M6024↓_LOG紀錄 秒-2
D20415  ; M6024↓_LOG紀錄 月-3
D20416  ; M6024↓_LOG紀錄 日-3
D20417  ; M6024↓_LOG紀錄 時-3
D20418  ; M6024↓_LOG紀錄 分-3
D20419  ; M6024↓_LOG紀錄 秒-3
D20421  ; M6025↑_LOG紀錄 日-1
D20422  ; M6025↑_LOG紀錄 時-1
D20423  ; M6025↑_LOG紀錄 分-1
D20424  ; M6025↑_LOG紀錄 秒-1
D20426  ; M6025↑_LOG紀錄 日-2
D20427  ; M6025↑_LOG紀錄 時-2
D20428  ; M6025↑_LOG紀錄 分-2
D20429  ; M6025↑_LOG紀錄 秒-2
D20430  ; M6025↑_LOG紀錄 月-3
D20431  ; M6025↑_LOG紀錄 日-3
D20432  ; M6025↑_LOG紀錄 時-3
D20433  ; M6025↑_LOG紀錄 分-3
D20434  ; M6025↑_LOG紀錄 秒-3
D20436  ; M6025↓_LOG紀錄 日-1
D20437  ; M6025↓_LOG紀錄 時-1
D20438  ; M6025↓_LOG紀錄 分-1
D20439  ; M6025↓_LOG紀錄 秒-1
D20441  ; M6025↓_LOG紀錄 日-2
D20442  ; M6025↓_LOG紀錄 時-2
D20443  ; M6025↓_LOG紀錄 分-2
D20444  ; M6025↓_LOG紀錄 秒-2
D20445  ; M6025↓_LOG紀錄 月-3
D20446  ; M6025↓_LOG紀錄 日-3
D20447  ; M6025↓_LOG紀錄 時-3
D20448  ; M6025↓_LOG紀錄 分-3
D20449  ; M6025↓_LOG紀錄 秒-3
D20451  ; M6105↑_LOG紀錄 日-1
D20452  ; M6105↑_LOG紀錄 時-1
D20453  ; M6105↑_LOG紀錄 分-1
D20454  ; M6105↑_LOG紀錄 秒-1
D20456  ; M6105↑_LOG紀錄 日-2
D20457  ; M6105↑_LOG紀錄 時-2
D20458  ; M6105↑_LOG紀錄 分-2
D20459  ; M6105↑_LOG紀錄 秒-2
D20460  ; M6105↑_LOG紀錄 月-3
D20461  ; M6105↑_LOG紀錄 日-3
D20462  ; M6105↑_LOG紀錄 時-3
D20463  ; M6105↑_LOG紀錄 分-3
D20464  ; M6105↑_LOG紀錄 秒-3
D20466  ; M6105↓_LOG紀錄 日-1
D20467  ; M6105↓_LOG紀錄 時-1
D20468  ; M6105↓_LOG紀錄 分-1
D20469  ; M6105↓_LOG紀錄 秒-1
D20471  ; M6105↓_LOG紀錄 日-2
D20472  ; M6105↓_LOG紀錄 時-2
D20473  ; M6105↓_LOG紀錄 分-2
D20474  ; M6105↓_LOG紀錄 秒-2
D20475  ; M6105↓_LOG紀錄 月-3
D20476  ; M6105↓_LOG紀錄 日-3
D20477  ; M6105↓_LOG紀錄 時-3
D20478  ; M6105↓_LOG紀錄 分-3
D20479  ; M6105↓_LOG紀錄 秒-3
D20481  ; M6106↑_LOG紀錄 日-1
D20482  ; M6106↑_LOG紀錄 時-1
D20483  ; M6106↑_LOG紀錄 分-1
D20484  ; M6106↑_LOG紀錄 秒-1
D20486  ; M6106↑_LOG紀錄 日-2
D20487  ; M6106↑_LOG紀錄 時-2
D20488  ; M6106↑_LOG紀錄 分-2
D20489  ; M6106↑_LOG紀錄 秒-2
D20490  ; M6106↑_LOG紀錄 月-3
D20491  ; M6106↑_LOG紀錄 日-3
D20492  ; M6106↑_LOG紀錄 時-3
D20493  ; M6106↑_LOG紀錄 分-3
D20494  ; M6106↑_LOG紀錄 秒-3
D20496  ; M6106↓_LOG紀錄 日-1
D20497  ; M6106↓_LOG紀錄 時-1
D20498  ; M6106↓_LOG紀錄 分-1
D20499  ; M6106↓_LOG紀錄 秒-1
D20501  ; M6106↓_LOG紀錄 日-2
D20502  ; M6106↓_LOG紀錄 時-2
D20503  ; M6106↓_LOG紀錄 分-2
D20504  ; M6106↓_LOG紀錄 秒-2
D20505  ; M6106↓_LOG紀錄 月-3
D20506  ; M6106↓_LOG紀錄 日-3
D20507  ; M6106↓_LOG紀錄 時-3
D20508  ; M6106↓_LOG紀錄 分-3
D20509  ; M6106↓_LOG紀錄 秒-3
D20511  ; M6107↑_LOG紀錄 日-1
D20512  ; M6107↑_LOG紀錄 時-1
D20513  ; M6107↑_LOG紀錄 分-1
D20514  ; M6107↑_LOG紀錄 秒-1
D20516  ; M6107↑_LOG紀錄 日-2
D20517  ; M6107↑_LOG紀錄 時-2
D20518  ; M6107↑_LOG紀錄 分-2
D20519  ; M6107↑_LOG紀錄 秒-2
D20520  ; M6107↑_LOG紀錄 月-3
D20521  ; M6107↑_LOG紀錄 日-3
D20522  ; M6107↑_LOG紀錄 時-3
D20523  ; M6107↑_LOG紀錄 分-3
D20524  ; M6107↑_LOG紀錄 秒-3
D20526  ; M6107↓_LOG紀錄 日-1
D20527  ; M6107↓_LOG紀錄 時-1
D20528  ; M6107↓_LOG紀錄 分-1
D20529  ; M6107↓_LOG紀錄 秒-1
D20531  ; M6107↓_LOG紀錄 日-2
D20532  ; M6107↓_LOG紀錄 時-2
D20533  ; M6107↓_LOG紀錄 分-2
D20534  ; M6107↓_LOG紀錄 秒-2
D20535  ; M6107↓_LOG紀錄 月-3
D20536  ; M6107↓_LOG紀錄 日-3
D20537  ; M6107↓_LOG紀錄 時-3
D20538  ; M6107↓_LOG紀錄 分-3
D20539  ; M6107↓_LOG紀錄 秒-3
D20541  ; M6056↑_LOG紀錄 日-1
D20542  ; M6056↑_LOG紀錄 時-1
D20543  ; M6056↑_LOG紀錄 分-1
D20544  ; M6056↑_LOG紀錄 秒-1
D20546  ; M6056↑_LOG紀錄 日-2
D20547  ; M6056↑_LOG紀錄 時-2
D20548  ; M6056↑_LOG紀錄 分-2
D20549  ; M6056↑_LOG紀錄 秒-2
D20550  ; M6056↑_LOG紀錄 月-3
D20551  ; M6056↑_LOG紀錄 日-3
D20552  ; M6056↑_LOG紀錄 時-3
D20553  ; M6056↑_LOG紀錄 分-3
D20554  ; M6056↑_LOG紀錄 秒-3
D20556  ; M6056↓_LOG紀錄 日-1
D20557  ; M6056↓_LOG紀錄 時-1
D20558  ; M6056↓_LOG紀錄 分-1
D20559  ; M6056↓_LOG紀錄 秒-1
D20561  ; M6056↓_LOG紀錄 日-2
D20562  ; M6056↓_LOG紀錄 時-2
D20563  ; M6056↓_LOG紀錄 分-2
D20564  ; M6056↓_LOG紀錄 秒-2
D20565  ; M6056↓_LOG紀錄 月-3
D20566  ; M6056↓_LOG紀錄 日-3
D20567  ; M6056↓_LOG紀錄 時-3
D20568  ; M6056↓_LOG紀錄 分-3
D20569  ; M6056↓_LOG紀錄 秒-3
D20571  ; M6058↑_LOG紀錄 日-1
D20572  ; M6058↑_LOG紀錄 時-1
D20573  ; M6058↑_LOG紀錄 分-1
D20574  ; M6058↑_LOG紀錄 秒-1
D20576  ; M6058↑_LOG紀錄 日-2
D20577  ; M6058↑_LOG紀錄 時-2
D20578  ; M6058↑_LOG紀錄 分-2
D20579  ; M6058↑_LOG紀錄 秒-2
D20580  ; M6058↑_LOG紀錄 月-3
D20581  ; M6058↑_LOG紀錄 日-3
D20582  ; M6058↑_LOG紀錄 時-3
D20583  ; M6058↑_LOG紀錄 分-3
D20584  ; M6058↑_LOG紀錄 秒-3
D20586  ; M6058↓_LOG紀錄 日-1
D20587  ; M6058↓_LOG紀錄 時-1
D20588  ; M6058↓_LOG紀錄 分-1
D20589  ; M6058↓_LOG紀錄 秒-1
D20591  ; M6058↓_LOG紀錄 日-2
D20592  ; M6058↓_LOG紀錄 時-2
D20593  ; M6058↓_LOG紀錄 分-2
D20594  ; M6058↓_LOG紀錄 秒-2
D20595  ; M6058↓_LOG紀錄 月-3
D20596  ; M6058↓_LOG紀錄 日-3
D20597  ; M6058↓_LOG紀錄 時-3
D20598  ; M6058↓_LOG紀錄 分-3
D20599  ; M6058↓_LOG紀錄 秒-3
D20601  ; M6104↑_LOG紀錄 日-1
D20602  ; M6104↑_LOG紀錄 時-1
D20603  ; M6104↑_LOG紀錄 分-1
D20604  ; M6104↑_LOG紀錄 秒-1
D20606  ; M6104↑_LOG紀錄 日-2
D20607  ; M6104↑_LOG紀錄 時-2
D20608  ; M6104↑_LOG紀錄 分-2
D20609  ; M6104↑_LOG紀錄 秒-2
D20610  ; M6104↑_LOG紀錄 月-3
D20611  ; M6104↑_LOG紀錄 日-3
D20612  ; M6104↑_LOG紀錄 時-3
D20613  ; M6104↑_LOG紀錄 分-3
D20614  ; M6104↑_LOG紀錄 秒-3
D20616  ; M6104↓_LOG紀錄 日-1
D20617  ; M6104↓_LOG紀錄 時-1
D20618  ; M6104↓_LOG紀錄 分-1
D20619  ; M6104↓_LOG紀錄 秒-1
D20621  ; M6104↓_LOG紀錄 日-2
D20622  ; M6104↓_LOG紀錄 時-2
D20623  ; M6104↓_LOG紀錄 分-2
D20624  ; M6104↓_LOG紀錄 秒-2
D20625  ; M6104↓_LOG紀錄 月-3
D20626  ; M6104↓_LOG紀錄 日-3
D20627  ; M6104↓_LOG紀錄 時-3
D20628  ; M6104↓_LOG紀錄 分-3
D20629  ; M6104↓_LOG紀錄 秒-3
D20631  ; M6042↑_LOG紀錄 日-1
D20632  ; M6042↑_LOG紀錄 時-1
D20633  ; M6042↑_LOG紀錄 分-1
D20634  ; M6042↑_LOG紀錄 秒-1
D20636  ; M6042↑_LOG紀錄 日-2
D20637  ; M6042↑_LOG紀錄 時-2
D20638  ; M6042↑_LOG紀錄 分-2
D20639  ; M6042↑_LOG紀錄 秒-2
D20640  ; M6042↑_LOG紀錄 月-3
D20641  ; M6042↑_LOG紀錄 日-3
D20642  ; M6042↑_LOG紀錄 時-3
D20643  ; M6042↑_LOG紀錄 分-3
D20644  ; M6042↑_LOG紀錄 秒-3
D20646  ; M6042↓_LOG紀錄 日-1
D20647  ; M6042↓_LOG紀錄 時-1
D20648  ; M6042↓_LOG紀錄 分-1
D20649  ; M6042↓_LOG紀錄 秒-1
D20651  ; M6042↓_LOG紀錄 日-2
D20652  ; M6042↓_LOG紀錄 時-2
D20653  ; M6042↓_LOG紀錄 分-2
D20654  ; M6042↓_LOG紀錄 秒-2
D20655  ; M6042↓_LOG紀錄 月-3
D20656  ; M6042↓_LOG紀錄 日-3
D20657  ; M6042↓_LOG紀錄 時-3
D20658  ; M6042↓_LOG紀錄 分-3
D20659  ; M6042↓_LOG紀錄 秒-3
D20661  ; M6043↑_LOG紀錄 日-1
D20662  ; M6043↑_LOG紀錄 時-1
D20663  ; M6043↑_LOG紀錄 分-1
D20664  ; M6043↑_LOG紀錄 秒-1
D20666  ; M6043↑_LOG紀錄 日-2
D20667  ; M6043↑_LOG紀錄 時-2
D20668  ; M6043↑_LOG紀錄 分-2
D20669  ; M6043↑_LOG紀錄 秒-2
D20670  ; M6043↑_LOG紀錄 月-3
D20671  ; M6043↑_LOG紀錄 日-3
D20672  ; M6043↑_LOG紀錄 時-3
D20673  ; M6043↑_LOG紀錄 分-3
D20674  ; M6043↑_LOG紀錄 秒-3
D20676  ; M6043↓_LOG紀錄 日-1
D20677  ; M6043↓_LOG紀錄 時-1
D20678  ; M6043↓_LOG紀錄 分-1
D20679  ; M6043↓_LOG紀錄 秒-1
D20681  ; M6043↓_LOG紀錄 日-2
D20682  ; M6043↓_LOG紀錄 時-2
D20683  ; M6043↓_LOG紀錄 分-2
D20684  ; M6043↓_LOG紀錄 秒-2
D20685  ; M6043↓_LOG紀錄 月-3
D20686  ; M6043↓_LOG紀錄 日-3
D20687  ; M6043↓_LOG紀錄 時-3
D20688  ; M6043↓_LOG紀錄 分-3
D20689  ; M6043↓_LOG紀錄 秒-3
D20691  ; M6111↑_LOG紀錄 日-1
D20692  ; M6111↑_LOG紀錄 時-1
D20693  ; M6111↑_LOG紀錄 分-1
D20694  ; M6111↑_LOG紀錄 秒-1
D20696  ; M6111↑_LOG紀錄 日-2
D20697  ; M6111↑_LOG紀錄 時-2
D20698  ; M6111↑_LOG紀錄 分-2
D20699  ; M6111↑_LOG紀錄 秒-2
D20700  ; M6111↑_LOG紀錄 月-3
D20701  ; M6111↑_LOG紀錄 日-3
D20702  ; M6111↑_LOG紀錄 時-3
D20703  ; M6111↑_LOG紀錄 分-3
D20704  ; M6111↑_LOG紀錄 秒-3
D20706  ; M6111↓_LOG紀錄 日-1
D20707  ; M6111↓_LOG紀錄 時-1
D20708  ; M6111↓_LOG紀錄 分-1
D20709  ; M6111↓_LOG紀錄 秒-1
D20711  ; M6111↓_LOG紀錄 日-2
D20712  ; M6111↓_LOG紀錄 時-2
D20713  ; M6111↓_LOG紀錄 分-2
D20714  ; M6111↓_LOG紀錄 秒-2
D20715  ; M6111↓_LOG紀錄 月-3
D20716  ; M6111↓_LOG紀錄 日-3
D20717  ; M6111↓_LOG紀錄 時-3
D20718  ; M6111↓_LOG紀錄 分-3
D20719  ; M6111↓_LOG紀錄 秒-3
D20721  ; M6112↑_LOG紀錄 日-1
D20722  ; M6112↑_LOG紀錄 時-1
D20723  ; M6112↑_LOG紀錄 分-1
D20724  ; M6112↑_LOG紀錄 秒-1
D20726  ; M6112↑_LOG紀錄 日-2
D20727  ; M6112↑_LOG紀錄 時-2
D20728  ; M6112↑_LOG紀錄 分-2
D20729  ; M6112↑_LOG紀錄 秒-2
D20730  ; M6112↑_LOG紀錄 月-3
D20731  ; M6112↑_LOG紀錄 日-3
D20732  ; M6112↑_LOG紀錄 時-3
D20733  ; M6112↑_LOG紀錄 分-3
D20734  ; M6112↑_LOG紀錄 秒-3
D20736  ; M6112↓_LOG紀錄 日-1
D20737  ; M6112↓_LOG紀錄 時-1
D20738  ; M6112↓_LOG紀錄 分-1
D20739  ; M6112↓_LOG紀錄 秒-1
D20741  ; M6112↓_LOG紀錄 日-2
D20742  ; M6112↓_LOG紀錄 時-2
D20743  ; M6112↓_LOG紀錄 分-2
D20744  ; M6112↓_LOG紀錄 秒-2
D20745  ; M6112↓_LOG紀錄 月-3
D20746  ; M6112↓_LOG紀錄 日-3
D20747  ; M6112↓_LOG紀錄 時-3
D20748  ; M6112↓_LOG紀錄 分-3
D20749  ; M6112↓_LOG紀錄 秒-3
D20751  ; M6006↑_LOG紀錄 日-1
D20752  ; M6006↑_LOG紀錄 時-1
D20753  ; M6006↑_LOG紀錄 分-1
D20754  ; M6006↑_LOG紀錄 秒-1
D20756  ; M6006↑_LOG紀錄 日-2
D20757  ; M6006↑_LOG紀錄 時-2
D20758  ; M6006↑_LOG紀錄 分-2
D20759  ; M6006↑_LOG紀錄 秒-2
D20760  ; M6006↑_LOG紀錄 月-3
D20761  ; M6006↑_LOG紀錄 日-3
D20762  ; M6006↑_LOG紀錄 時-3
D20763  ; M6006↑_LOG紀錄 分-3
D20764  ; M6006↑_LOG紀錄 秒-3
D20766  ; M6006↓_LOG紀錄 日-1
D20767  ; M6006↓_LOG紀錄 時-1
D20768  ; M6006↓_LOG紀錄 分-1
D20769  ; M6006↓_LOG紀錄 秒-1
D20771  ; M6006↓_LOG紀錄 日-2
D20772  ; M6006↓_LOG紀錄 時-2
D20773  ; M6006↓_LOG紀錄 分-2
D20774  ; M6006↓_LOG紀錄 秒-2
D20775  ; M6006↓_LOG紀錄 月-3
D20776  ; M6006↓_LOG紀錄 日-3
D20777  ; M6006↓_LOG紀錄 時-3
D20778  ; M6006↓_LOG紀錄 分-3
D20779  ; M6006↓_LOG紀錄 秒-3
D21002  ; D9105↑_LOG紀錄 日-1
D21003  ; D9105↑_LOG紀錄 時-1
D21004  ; D9105↑_LOG紀錄 分-1
D21005  ; D9105↑_LOG紀錄 秒-1
D21007  ; D9105↑_LOG紀錄 月-2
D21008  ; D9105↑_LOG紀錄 日-2
D21009  ; D9105↑_LOG紀錄 時-2
D21010  ; D9105↑_LOG紀錄 分-2
D21011  ; D9105↑_LOG紀錄 秒-2
D21012  ; D9105↑_LOG紀錄 值-3
D21013  ; D9105↑_LOG紀錄 月-3
D21014  ; D9105↑_LOG紀錄 日-3
D21015  ; D9105↑_LOG紀錄 時-3
D21016  ; D9105↑_LOG紀錄 分-3
D21017  ; D9105↑_LOG紀錄 秒-3
D21018  ; D9105↑_LOG紀錄 值-4
D21019  ; D9105↑_LOG紀錄 月-4
D21020  ; D9105↑_LOG紀錄 日-4
D21021  ; D9105↑_LOG紀錄 時-4
D21022  ; D9105↑_LOG紀錄 分-4
D21023  ; D9105↑_LOG紀錄 秒-4
D21024  ; D9105↑_LOG紀錄 值-5
D21025  ; D9105↑_LOG紀錄 月-5
D21026  ; D9105↑_LOG紀錄 日-5
D21027  ; D9105↑_LOG紀錄 時-5
D21028  ; D9105↑_LOG紀錄 分-5
D21029  ; D9105↑_LOG紀錄 秒-5
D21032  ; D9099↑_LOG紀錄 日-1
D21033  ; D9099↑_LOG紀錄 時-1
D21034  ; D9099↑_LOG紀錄 分-1
D21035  ; D9099↑_LOG紀錄 秒-1
D21037  ; D9099↑_LOG紀錄 月-2
D21038  ; D9099↑_LOG紀錄 日-2
D21039  ; D9099↑_LOG紀錄 時-2
D21040  ; D9099↑_LOG紀錄 分-2
D21041  ; D9099↑_LOG紀錄 秒-2
D21042  ; D9099↑_LOG紀錄 值-3
D21043  ; D9099↑_LOG紀錄 月-3
D21044  ; D9099↑_LOG紀錄 日-3
D21045  ; D9099↑_LOG紀錄 時-3
D21046  ; D9099↑_LOG紀錄 分-3
D21047  ; D9099↑_LOG紀錄 秒-3
D21048  ; D9099↑_LOG紀錄 值-4
D21049  ; D9099↑_LOG紀錄 月-4
D21050  ; D9099↑_LOG紀錄 日-4
D21051  ; D9099↑_LOG紀錄 時-4
D21052  ; D9099↑_LOG紀錄 分-4
D21053  ; D9099↑_LOG紀錄 秒-4
D21054  ; D9099↑_LOG紀錄 值-5
D21055  ; D9099↑_LOG紀錄 月-5
D21056  ; D9099↑_LOG紀錄 日-5
D21057  ; D9099↑_LOG紀錄 時-5
D21058  ; D9099↑_LOG紀錄 分-5
D21059  ; D9099↑_LOG紀錄 秒-5
W103  ; 1槽風速CH5顯示
W104  ; 2槽風速CH6顯示
W105  ; 3槽風速CH7顯示
W106  ; 4槽風速CH8顯示
W107  ; 5槽風速CH9顯示
W10C  ; 1靜置風速顯示
W10D  ; 2靜置風速顯示
W10E  ; 1冷卻風速CH10轉顯示
W10F  ; 2冷卻風速CH11顯示
R1000  ; PASSWORELEVEL 01
R1001  ; PASSWORELEVEL 01
R1002  ; PASSWORELEVEL 02
R1003  ; PASSWORELEVEL 02
R1004  ; PASSWORELEVEL 03
R1005  ; PASSWORELEVEL 03
R1006  ; PASSWORELEVEL 04
R1007  ; PASSWORELEVEL 04
R1008  ; PASSWORELEVEL 05
R1009  ; PASSWORELEVEL 05
R1010  ; PASSWORELEVEL 06
R1011  ; PASSWORELEVEL 06
R1012  ; PASSWORELEVEL 07
R1013  ; PASSWORELEVEL 07
R1014  ; PASSWORELEVEL 08
R1015  ; PASSWORELEVEL 08
R1016  ; PASSWORELEVEL 09
R1017  ; PASSWORELEVEL 09
R1018  ; PASSWORELEVEL 10
R1019  ; PASSWORELEVEL 10
R1020  ; PASSWORELEVEL 11
R1021  ; PASSWORELEVEL 11
R1022  ; PASSWORELEVEL 12
R1023  ; PASSWORELEVEL 12
R1024  ; PASSWORELEVEL 13
R1025  ; PASSWORELEVEL 13
R1026  ; PASSWORELEVEL 14
R1027  ; PASSWORELEVEL 14
R1028  ; PASSWORELEVEL 15
R1029  ; PASSWORELEVEL 15
R6000  ; 板架計數
ZR0  ; [ED-02] Modify Type
ZR1  ; [ED-02] RecipeID#02/01
ZR2  ; [ED-02] RecipeID#04/03
ZR3  ; [ED-02] RecipeID#06/05
ZR4  ; [ED-02] RecipeID#08/07
ZR5  ; [ED-02] RecipeID#10/09
ZR6  ; [ED-02] RecipeID#12/11
ZR7  ; [ED-02] RecipeID#14/13
ZR8  ; [ED-02] RecipeID#16/15
ZR9  ; [ED-02] RecipeID#18/17
ZR10  ; [ED-02] RecipeID#20/19
ZR11  ; [ED-02] RecipeID#22/21
ZR12  ; [ED-02] RecipeID#24/23
ZR13  ; [ED-02] RecipeID#26/25
ZR14  ; [ED-02] RecipeID#28/27
ZR15  ; [ED-02] RecipeID#30/29
ZR21  ; [ED-02] HEAT-SV #01
ZR22  ; [ED-02] HEAT-SV #02
ZR23  ; [ED-02] HEAT-SV #03
ZR24  ; [ED-02] HEAT-SV #04
ZR25  ; [ED-02] HEAT-SV #05
ZR26  ; [ED-02] HEAT-SV #06
ZR27  ; [ED-02] HEAT-SV #07
ZR28  ; [ED-02] HEAT-SV #08
ZR29  ; [ED-02] HEAT-SV #09
ZR30  ; [ED-02] HEAT-SV #10
ZR31  ; [ED-02] HEAT-SV #11
ZR32  ; [ED-02] HEAT-SV #12
ZR146  ; 上報軟體編號SoftRev
ZR147  ; 上報軟體編號SoftRev
ZR151  ; Code-S7-F23-F25
ZR157  ; 上報儲存配方處理0=OK,3=沒空間
ZR2035  ; SECS_上位下載配方Recipe NO.
ZR2036  ; SECS_上位下載配方RecipeID#02/01
ZR2037  ; SECS_上位下載配方RecipeID#04/03
ZR2038  ; SECS_上位下載配方RecipeID#06/05
ZR2039  ; SECS_上位下載配方RecipeID#08/07
ZR2040  ; SECS_上位下載配方RecipeID#10/09
ZR2041  ; SECS_上位下載配方RecipeID#12/11
ZR2042  ; SECS_上位下載配方RecipeID#14/13
ZR2043  ; SECS_上位下載配方RecipeID#16/15
ZR2044  ; SECS_上位下載配方RecipeID#18/17
ZR2045  ; SECS_上位下載配方RecipeID#20/19
ZR2046  ; SECS_上位下載配方第01槽電熱設定
ZR2047  ; SECS_上位下載配方第02槽電熱設定
ZR2048  ; SECS_上位下載配方第03槽電熱設定
ZR2049  ; SECS_上位下載配方第04槽電熱設定
ZR2050  ; SECS_上位下載配方第05槽電熱設定
ZR2051  ; SECS_上位下載配方第06槽電熱設定
ZR2052  ; SECS_上位下載配方第07槽電熱設定
ZR2053  ; SECS_上位下載配方第08槽電熱設定
ZR2054  ; SECS_上位下載配方第09槽電熱設定
ZR2055  ; SECS_上位下載配方第10槽電熱設定
ZR2056  ; SECS_上位下載配方第11槽電熱設定
ZR2057  ; SECS_上位下載配方第12槽電熱設定
ZR2058  ; SECS_上位下載配方進料步進間隔次
ZR2059  ; SECS_上位下載配方烘烤步進時間設
ZR2060  ; SECS_上位下載配方板材尺寸寬度設
ZR5201  ; SECS_上位配方NO.01
ZR5299  ; SECS_上位配方NO.50
ZR10001  ; 異動暫存RecipeID#02/01
ZR10002  ; 異動暫存RecipeID#04/03
ZR10003  ; 異動暫存RecipeID#06/05
ZR10004  ; 異動暫存RecipeID#08/07
ZR10005  ; 異動暫存RecipeID#10/09
ZR10006  ; 異動暫存RecipeID#12/11
ZR10007  ; 異動暫存RecipeID#14/13
ZR10008  ; 異動暫存RecipeID#16/15
ZR10009  ; 異動暫存RecipeID#18/17
ZR10010  ; 異動暫存RecipeID#20/19
ZR10011  ; 異動暫存RecipeID#22/21
ZR10012  ; 異動暫存RecipeID#24/23
ZR10013  ; 異動暫存RecipeID#26/25
ZR10014  ; 異動暫存RecipeID#28/27
ZR10015  ; 異動暫存RecipeID#30/29
ZR10016  ; 異動暫存RecipeID#32/31
ZR10017  ; 異動暫存RecipeID#34/33
ZR10018  ; 異動暫存RecipeID#36/35
ZR10019  ; 異動暫存RecipeID#38/37
ZR10020  ; 異動暫存RecipeID#40/39
ZR10021  ; 異動暫存第01槽電熱設定
ZR10022  ; 異動暫存第02槽電熱設定
ZR10023  ; 異動暫存第03槽電熱設定
ZR10024  ; 異動暫存第04槽電熱設定
ZR10025  ; 異動暫存第05槽電熱設定
ZR10026  ; 異動暫存第06槽電熱設定
ZR10027  ; 異動暫存第07槽電熱設定
ZR10028  ; 異動暫存第08槽電熱設定
ZR10029  ; 異動暫存第09槽電熱設定
ZR10030  ; 異動暫存第10槽電熱設定
ZR10031  ; 異動暫存第11槽電熱設定
ZR10032  ; 異動暫存第12槽電熱設定
ZR10033  ; 異動暫存進料步進間隔次數設定
ZR10034  ; 異動暫存烘烤步進時間設定
ZR10035  ; 異動暫存板材尺寸寬度設定
ZR10039  ; 異動暫存烘烤時間(分)
P0  ; 初始設定
P5  ; 功能選擇
P10  ; FX2N-2AD
P20  ; FX2N-1PG(昇降)
P90  ; 原點訊號
P100  ; 進料機構
P105  ; 上料機構
P110  ; 下料機構
P120  ; 下料位移機構
P130  ; 電熱啟動停止
P140  ; 風車電熱訊號
P150  ; 產能履歷
P160  ; 設備運轉保養時間
P170  ; 電熱風車異常訊號
P180  ; 一般異常
P190  ; 烘烤時間
D5002.0  ; GP->ATMA_ROBOT準備取板
D5002.1  ; GP->ATMA_ROBOT動作完成
D5102.8  ; ATMA->GP_印刷機連線
D5102.9  ; ATMA->GP_印刷機取板要求
D5102.A  ; ATMA->GP_印刷機動作異常
